LIN {X 0,Y 150.229,Z 301.582,A -85,B 0,C 180,E1 -24092.731,E2 -24092.731} C_VEL
LIN {X 0,Y 150.411,Z 301.529,A -85,B 0,C 180,E1 -24099.15,E2 -24099.15} C_VEL
LIN {X 0,Y 151.251,Z 301.453,A -85,B 0,C 180,E1 -24104.699,E2 -24104.699} C_VEL
LIN {X 0,Y 152.579,Z 314.488,A -85,B 0,C 180,E1 -24105.834,E2 -24105.834} C_VEL
LIN {X 0,Y 152.143,Z 366.9,A -85,B 0,C 180,E1 -24110.789,E2 -24110.789} C_VEL
LIN {X 0,Y 151.908,Z 379.421,A -85,B 0,C 180,E1 -24112.365,E2 -24112.365} C_VEL
LIN {X 0,Y 151.505,Z 390.839,A -85,B 0,C 180,E1 -24114.352,E2 -24114.352} C_VEL
LIN {X 0,Y 151.14,Z 401.236,A -85,B 0,C 180,E1 -24116.677,E2 -24116.677} C_VEL
LIN {X 0,Y 150.848,Z 410.602,A -85,B 0,C 180,E1 -24119.341,E2 -24119.341} C_VEL
LIN {X 0,Y 150.628,Z 416.487,A -85,B 0,C 180,E1 -24121.345,E2 -24121.345} C_VEL
LIN {X 0,Y 150.402,Z 424.552,A -85,B 0,C 180,E1 -24124.699,E2 -24124.699} C_VEL
LIN {X 0,Y 150.691,Z 431.338,A -85,B 0,C 180,E1 -24128.051,E2 -24128.051} C_VEL
LIN {X 0,Y 151.578,Z 437.961,A -85,B 0,C 180,E1 -24132.051,E2 -24132.051} C_VEL
LIN {X 0,Y 153.375,Z 443.251,A -85,B 0,C 180,E1 -24135.966,E2 -24135.966} C_VEL
LIN {X 0,Y 156.284,Z 447.464,A -85,B 0,C 180,E1 -24139.719,E2 -24139.719} C_VEL
LIN {X 0,Y 160.116,Z 450.667,A -85,B 0,C 180,E1 -24143.276,E2 -24143.276} C_VEL
LIN {X 0,Y 163.094,Z 452.341,A -85,B 0,C 180,E1 -24145.534,E2 -24145.534} C_VEL
LIN {X 0,Y 168.824,Z 454.022,A -85,B 0,C 180,E1 -24149.047,E2 -24149.047} C_VEL
LIN {X 0,Y 174.154,Z 454.577,A -85,B 0,C 180,E1 -24151.65,E2 -24151.65} C_VEL
LIN {X 0,Y 178.432,Z 454.52,A -85,B 0,C 180,E1 -24153.472,E2 -24153.472} C_VEL
LIN {X 0,Y 182.969,Z 453.929,A -85,B 0,C 180,E1 -24155.188,E2 -24155.188} C_VEL
LIN {X 0,Y 192.773,Z 451.539,A -85,B 0,C 180,E1 -24158.307,E2 -24158.307} C_VEL
LIN {X 0,Y 200.616,Z 448.43,A -85,B 0,C 180,E1 -24160.405,E2 -24160.405} C_VEL
LIN {X 0,Y 208.853,Z 444.151,A -85,B 0,C 180,E1 -24162.306,E2 -24162.306} C_VEL
LIN {X 0,Y 216.089,Z 439.514,A -85,B 0,C 180,E1 -24163.759,E2 -24163.759} C_VEL
LIN {X 0,Y 217.224,Z 438.727,A -85,B 0,C 180,E1 -24163.963,E2 -24163.963} C_VEL
LIN {X 0,Y 216.329,Z 439.432,A -85,B 0,C 180,E1 -24164.379,E2 -24164.379} C_VEL
LIN {X 0,Y 210.261,Z 443.858,A -85,B 0,C 180,E1 -24165.417,E2 -24165.417} C_VEL
LIN {X 0,Y 202.4,Z 448.708,A -85,B 0,C 180,E1 -24166.984,E2 -24166.984} C_VEL
LIN {X 0,Y 193.364,Z 453.242,A -85,B 0,C 180,E1 -24169.138,E2 -24169.138} C_VEL
LIN {X 0,Y 185.87,Z 456.12,A -85,B 0,C 180,E1 -24171.275,E2 -24171.275} C_VEL
LIN {X 0,Y 178.466,Z 458.224,A -85,B 0,C 180,E1 -24173.793,E2 -24173.793} C_VEL
LIN {X 0,Y 172.785,Z 459.125,A -85,B 0,C 180,E1 -24176.161,E2 -24176.161} C_VEL
LIN {X 0,Y 168.905,Z 459.398,A -85,B 0,C 180,E1 -24177.655,E2 -24177.655} C_VEL
LIN {X 0,Y 164.5,Z 459.233,A -85,B 0,C 180,E1 -24179.027,E2 -24179.027} C_VEL
LIN {X 0,Y 157.202,Z 458.002,A -85,B 0,C 180,E1 -24181.38,E2 -24181.38} C_VEL
LIN {X 0,Y 152.596,Z 456.474,A -85,B 0,C 180,E1 -24183.671,E2 -24183.671} C_VEL
LIN {X 0,Y 151.792,Z 455.973,A -85,B 0,C 180,E1 -24184.331,E2 -24184.331} C_VEL
LIN {X 0,Y 148.796,Z 453.802,A -85,B 0,C 180,E1 -24187.798,E2 -24187.798} C_VEL
LIN {X 0,Y 145.917,Z 449.099,A -85,B 0,C 180,E1 -24193.202,E2 -24193.202} C_VEL
LIN {X 0,Y 145.117,Z 445.833,A -85,B 0,C 180,E1 -24196.344,E2 -24196.344} C_VEL
LIN {X 0,Y 143.265,Z 449.83,A -85,B 0,C 180,E1 -24198.683,E2 -24198.683} C_VEL
LIN {X 0,Y 141.516,Z 455.368,A -85,B 0,C 180,E1 -24202.867,E2 -24202.867} C_VEL
LIN {X 0,Y 141.005,Z 459.469,A -85,B 0,C 180,E1 -24207.142,E2 -24207.142} C_VEL
LIN {X 0,Y 141.109,Z 461.507,A -85,B 0,C 180,E1 -24209.999,E2 -24209.999} C_VEL
LIN {X 0,Y 140.819,Z 463.144,A -85,B 0,C 180,E1 -24213.359,E2 -24213.359} C_VEL
LIN {X 0,Y 140.801,Z 463.878,A -85,B 0,C 180,E1 -24215.729,E2 -24215.729} C_VEL
LIN {X 0,Y 141.059,Z 464.25,A -85,B 0,C 180,E1 -24218.596,E2 -24218.596} C_VEL
LIN {X 0,Y 141.652,Z 464.181,A -85,B 0,C 180,E1 -24221.446,E2 -24221.446} C_VEL
LIN {X 0,Y 142.592,Z 463.67,A -85,B 0,C 180,E1 -24224.266,E2 -24224.266} C_VEL
LIN {X 0,Y 143.865,Z 462.646,A -85,B 0,C 180,E1 -24227.044,E2 -24227.044} C_VEL
LIN {X 0,Y 146.436,Z 460.124,A -85,B 0,C 180,E1 -24231.097,E2 -24231.097} C_VEL
LIN {X 0,Y 149.84,Z 456.335,A -85,B 0,C 180,E1 -24234.969,E2 -24234.969} C_VEL
LIN {X 0,Y 153.97,Z 451.2,A -85,B 0,C 180,E1 -24238.637,E2 -24238.637} C_VEL
LIN {X 0,Y 157.929,Z 445.711,A -85,B 0,C 180,E1 -24241.526,E2 -24241.526} C_VEL
LIN {X 0,Y 162.256,Z 438.889,A -85,B 0,C 180,E1 -24244.269,E2 -24244.269} C_VEL
LIN {X 0,Y 166.858,Z 430.459,A -85,B 0,C 180,E1 -24246.751,E2 -24246.751} C_VEL
LIN {X 0,Y 170.617,Z 422.486,A -85,B 0,C 180,E1 -24248.537,E2 -24248.537} C_VEL
LIN {X 0,Y 173.829,Z 414.514,A -85,B 0,C 180,E1 -24249.928,E2 -24249.928} C_VEL
LIN {X 0,Y 176.671,Z 406.274,A -85,B 0,C 180,E1 -24251.023,E2 -24251.023} C_VEL
LIN {X 0,Y 179.008,Z 397.922,A -85,B 0,C 180,E1 -24251.869,E2 -24251.869} C_VEL
LIN {X 0,Y 180.963,Z 388.209,A -85,B 0,C 180,E1 -24252.618,E2 -24252.618} C_VEL
LIN {X 0,Y 182.34,Z 377.856,A -85,B 0,C 180,E1 -24253.135,E2 -24253.135} C_VEL
LIN {X 0,Y 182.818,Z 371.037,A -85,B 0,C 180,E1 -24253.41,E2 -24253.41} C_VEL
LIN {X 0,Y 182.252,Z 365.36,A -85,B 0,C 180,E1 -24253.978,E2 -24253.978} C_VEL
LIN {X 0,Y 177.633,Z 353.901,A -85,B 0,C 180,E1 -24256.616,E2 -24256.616} C_VEL
LIN {X 0,Y 173.526,Z 345.27,A -85,B 0,C 180,E1 -24259.122,E2 -24259.122} C_VEL
LIN {X 0,Y 170.096,Z 338.97,A -85,B 0,C 180,E1 -24261.374,E2 -24261.374} C_VEL
LIN {X 0,Y 167.541,Z 334.457,A -85,B 0,C 180,E1 -24263.23,E2 -24263.23} C_VEL
LIN {X 0,Y 165.381,Z 330.639,A -85,B 0,C 180,E1 -24264.943,E2 -24264.943} C_VEL
LIN {X 0,Y 162.264,Z 325.564,A -85,B 0,C 180,E1 -24267.65,E2 -24267.65} C_VEL
LIN {X 0,Y 158.625,Z 320.076,A -85,B 0,C 180,E1 -24271.317,E2 -24271.317} C_VEL
LIN {X 0,Y 155.794,Z 317.621,A -85,B 0,C 180,E1 -24274.531,E2 -24274.531} C_VEL
LIN {X 0,Y 154.29,Z 314.613,A -85,B 0,C 180,E1 -24276.858,E2 -24276.858} C_VEL
LIN {X 0,Y 150.682,Z 311.854,A -85,B 0,C 180,E1 -24284.088,E2 -24284.088} C_VEL
LIN {X 0,Y 149.696,Z 308.547,A -85,B 0,C 180,E1 -24290.37,E2 -24290.37} C_VEL
LIN {X 0,Y 149.797,Z 308.81,A -85,B 0,C 180,E1 -24294.607,E2 -24294.607} C_VEL
LIN {X 0,Y 150.803,Z 310.633,A -85,B 0,C 180,E1 -24299.491,E2 -24299.491} C_VEL
LIN {X 0,Y 152.574,Z 313.389,A -85,B 0,C 180,E1 -24303.953,E2 -24303.953} C_VEL
LIN {X 0,Y 154.674,Z 314.736,A -85,B 0,C 180,E1 -24307.333,E2 -24307.333} C_VEL
LIN {X 0,Y 156.305,Z 317.841,A -85,B 0,C 180,E1 -24309.747,E2 -24309.747} C_VEL
LIN {X 0,Y 158.766,Z 320.202,A -85,B 0,C 180,E1 -24312.506,E2 -24312.506} C_VEL
LIN {X 0,Y 161.046,Z 323.638,A -85,B 0,C 180,E1 -24314.864,E2 -24314.864} C_VEL
LIN {X 0,Y 162.738,Z 325.43,A -85,B 0,C 180,E1 -24316.364,E2 -24316.364} C_VEL
LIN {X 0,Y 165.495,Z 329.24,A -85,B 0,C 180,E1 -24318.67,E2 -24318.67} C_VEL
LIN {X 0,Y 169.55,Z 335.043,A -85,B 0,C 180,E1 -24321.669,E2 -24321.669} C_VEL
LIN {X 0,Y 174.099,Z 341.826,A -85,B 0,C 180,E1 -24324.579,E2 -24324.579} C_VEL
LIN {X 0,Y 179.901,Z 351.582,A -85,B 0,C 180,E1 -24327.867,E2 -24327.867} C_VEL
LIN {X 0,Y 183.667,Z 358.715,A -85,B 0,C 180,E1 -24329.822,E2 -24329.822} C_VEL
LIN {X 0,Y 182.291,Z 374.31,A -85,B 0,C 180,E1 -24330.493,E2 -24330.493} C_VEL
LIN {X 0,Y 180.442,Z 384.951,A -85,B 0,C 180,E1 -24331.303,E2 -24331.303} C_VEL
LIN {X 0,Y 178.509,Z 393.196,A -85,B 0,C 180,E1 -24332.171,E2 -24332.171} C_VEL
LIN {X 0,Y 175.887,Z 401.994,A -85,B 0,C 180,E1 -24333.392,E2 -24333.392} C_VEL
LIN {X 0,Y 172.716,Z 410.391,A -85,B 0,C 180,E1 -24334.863,E2 -24334.863} C_VEL
LIN {X 0,Y 169.499,Z 417.801,A -85,B 0,C 180,E1 -24336.549,E2 -24336.549} C_VEL
LIN {X 0,Y 166.077,Z 424.565,A -85,B 0,C 180,E1 -24338.476,E2 -24338.476} C_VEL
LIN {X 0,Y 161.746,Z 431.819,A -85,B 0,C 180,E1 -24341.083,E2 -24341.083} C_VEL
LIN {X 0,Y 157.132,Z 438.434,A -85,B 0,C 180,E1 -24344.306,E2 -24344.306} C_VEL
LIN {X 0,Y 154.039,Z 442.386,A -85,B 0,C 180,E1 -24346.872,E2 -24346.872} C_VEL
LIN {X 0,Y 151.295,Z 445.463,A -85,B 0,C 180,E1 -24349.434,E2 -24349.434} C_VEL
LIN {X 0,Y 148.822,Z 447.877,A -85,B 0,C 180,E1 -24352.128,E2 -24352.128} C_VEL
LIN {X 0,Y 146.718,Z 449.672,A -85,B 0,C 180,E1 -24354.914,E2 -24354.914} C_VEL
LIN {X 0,Y 144.872,Z 450.906,A -85,B 0,C 180,E1 -24357.75,E2 -24357.75} C_VEL
LIN {X 0,Y 142.605,Z 451.785,A -85,B 0,C 180,E1 -24362.486,E2 -24362.486} C_VEL
LIN {X 0,Y 141.321,Z 451.399,A -85,B 0,C 180,E1 -24366.557,E2 -24366.557} C_VEL
LIN {X 0,Y 140.573,Z 449.331,A -85,B 0,C 180,E1 -24371.754,E2 -24371.754} C_VEL
LIN {X 0,Y 140.589,Z 446.8,A -85,B 0,C 180,E1 -24375.526,E2 -24375.526} C_VEL
LIN {X 0,Y 141.098,Z 442.555,A -85,B 0,C 180,E1 -24379.961,E2 -24379.961} C_VEL
LIN {X 0,Y 142.197,Z 436.794,A -85,B 0,C 180,E1 -24384.328,E2 -24384.328} C_VEL
LIN {X 0,Y 143.366,Z 430.499,A -85,B 0,C 180,E1 -24387.894,E2 -24387.894} C_VEL
LIN {X 0,Y 144.639,Z 424.336,A -85,B 0,C 180,E1 -24390.697,E2 -24390.697} C_VEL
LIN {X 0,Y 146.197,Z 416.829,A -85,B 0,C 180,E1 -24393.446,E2 -24393.446} C_VEL
LIN {X 0,Y 147.588,Z 410.023,A -85,B 0,C 180,E1 -24395.466,E2 -24395.466} C_VEL
LIN {X 0,Y 149.047,Z 401.938,A -85,B 0,C 180,E1 -24397.415,E2 -24397.415} C_VEL
LIN {X 0,Y 150.452,Z 393.174,A -85,B 0,C 180,E1 -24399.071,E2 -24399.071} C_VEL
LIN {X 0,Y 151.565,Z 383.214,A -85,B 0,C 180,E1 -24400.521,E2 -24400.521} C_VEL
LIN {X 0,Y 152.71,Z 370.439,A -85,B 0,C 180,E1 -24401.707,E2 -24401.707} C_VEL
LIN {X 0,Y 153.76,Z 346.37,A -85,B 0,C 180,E1 -24402.886,E2 -24402.886} C_VEL
LIN {X 0,Y 154.41,Z 327.759,A -85,B 0,C 180,E1 -24403.733,E2 -24403.733} C_VEL
LIN {X 0,Y 150.233,Z 317.497,A -85,B 0,C 180,E1 -24404.997,E2 -24404.997} C_VEL
LIN {X 0,Y 144.242,Z 305.25,A -85,B 0,C 180,E1 -24406.817,E2 -24406.817} C_VEL
LIN {X 0,Y 143.241,Z 302.455,A -85,B 0,C 180,E1 -24407.213,E2 -24407.213} C_VEL
LIN {X 0,Y 143.249,Z 302.455,A -85,B 0,C 180,E1 -24411.256,E2 -24411.256} C_VEL
LIN {X 0,Y 143.159,Z 302.465,A -85,B 0,C 180,E1 -24417.936,E2 -24417.936} C_VEL
LIN {X 0,Y 143.113,Z 302.461,A -85,B 0,C 180,E1 -24423.421,E2 -24423.421} C_VEL
LIN {X 0,Y 143.032,Z 302.477,A -85,B 0,C 180,E1 -24429.701,E2 -24429.701} C_VEL
LIN {X 0,Y 143.014,Z 302.478,A -85,B 0,C 180,E1 -24433.472,E2 -24433.472} C_VEL
LIN {X 0,Y 143.022,Z 302.482,A -85,B 0,C 180,E1 -24437.485,E2 -24437.485} C_VEL
LIN {X 0,Y 143.06,Z 302.473,A -85,B 0,C 180,E1 -24441.816,E2 -24441.816} C_VEL
LIN {X 0,Y 143.164,Z 302.459,A -85,B 0,C 180,E1 -24447.329,E2 -24447.329} C_VEL
LIN {X 0,Y 143.146,Z 302.462,A -85,B 0,C 180,E1 -24453.788,E2 -24453.788} C_VEL
LIN {X 0,Y 143.414,Z 302.402,A -85,B 0,C 180,E1 -24459.948,E2 -24459.948} C_VEL
LIN {X 0,Y 144.372,Z 302.313,A -85,B 0,C 180,E1 -24465.33,E2 -24465.33} C_VEL
LIN {X 0,Y 145.649,Z 314.508,A -85,B 0,C 180,E1 -24466.404,E2 -24466.404} C_VEL
LIN {X 0,Y 145.428,Z 365.822,A -85,B 0,C 180,E1 -24471.586,E2 -24471.586} C_VEL
LIN {X 0,Y 145.209,Z 378.736,A -85,B 0,C 180,E1 -24473.234,E2 -24473.234} C_VEL
LIN {X 0,Y 144.862,Z 389.408,A -85,B 0,C 180,E1 -24475.139,E2 -24475.139} C_VEL
LIN {X 0,Y 144.515,Z 400.112,A -85,B 0,C 180,E1 -24477.57,E2 -24477.57} C_VEL
LIN {X 0,Y 144.262,Z 410.585,A -85,B 0,C 180,E1 -24480.707,E2 -24480.707} C_VEL
LIN {X 0,Y 143.969,Z 418.075,A -85,B 0,C 180,E1 -24483.507,E2 -24483.507} C_VEL
LIN {X 0,Y 143.94,Z 425.928,A -85,B 0,C 180,E1 -24487.02,E2 -24487.02} C_VEL
LIN {X 0,Y 144.613,Z 433.562,A -85,B 0,C 180,E1 -24491.218,E2 -24491.218} C_VEL
LIN {X 0,Y 146.4,Z 440.494,A -85,B 0,C 180,E1 -24495.958,E2 -24495.958} C_VEL
LIN {X 0,Y 148.706,Z 444.681,A -85,B 0,C 180,E1 -24499.327,E2 -24499.327} C_VEL
LIN {X 0,Y 152.233,Z 448.67,A -85,B 0,C 180,E1 -24503.113,E2 -24503.113} C_VEL
LIN {X 0,Y 156.758,Z 451.664,A -85,B 0,C 180,E1 -24506.645,E2 -24506.645} C_VEL
LIN {X 0,Y 163.972,Z 454.29,A -85,B 0,C 180,E1 -24510.961,E2 -24510.961} C_VEL
LIN {X 0,Y 172.553,Z 455.098,A -85,B 0,C 180,E1 -24514.773,E2 -24514.773} C_VEL
LIN {X 0,Y 177.248,Z 454.952,A -85,B 0,C 180,E1 -24516.503,E2 -24516.503} C_VEL
LIN {X 0,Y 182.189,Z 454.309,A -85,B 0,C 180,E1 -24518.12,E2 -24518.12} C_VEL
LIN {X 0,Y 187.345,Z 453.182,A -85,B 0,C 180,E1 -24519.63,E2 -24519.63} C_VEL
LIN {X 0,Y 198.186,Z 449.699,A -85,B 0,C 180,E1 -24522.366,E2 -24522.366} C_VEL
LIN {X 0,Y 203.871,Z 447.147,A -85,B 0,C 180,E1 -24523.594,E2 -24523.594} C_VEL
LIN {X 0,Y 205.328,Z 446.454,A -85,B 0,C 180,E1 -24524.044,E2 -24524.044} C_VEL
LIN {X 0,Y 195.558,Z 451.445,A -85,B 0,C 180,E1 -24525.96,E2 -24525.96} C_VEL
LIN {X 0,Y 188.075,Z 454.463,A -85,B 0,C 180,E1 -24527.729,E2 -24527.729} C_VEL
LIN {X 0,Y 182.737,Z 456.222,A -85,B 0,C 180,E1 -24529.17,E2 -24529.17} C_VEL
LIN {X 0,Y 172.779,Z 458.32,A -85,B 0,C 180,E1 -24532.399,E2 -24532.399} C_VEL
LIN {X 0,Y 167.077,Z 458.858,A -85,B 0,C 180,E1 -24534.749,E2 -24534.749} C_VEL
LIN {X 0,Y 160.228,Z 458.587,A -85,B 0,C 180,E1 -24538.24,E2 -24538.24} C_VEL
LIN {X 0,Y 156.703,Z 457.974,A -85,B 0,C 180,E1 -24540.439,E2 -24540.439} C_VEL
LIN {X 0,Y 151.792,Z 455.973,A -85,B 0,C 180,E1 -24544.331,E2 -24544.331} C_VEL
LIN {X 0,Y 149.289,Z 454.599,A -85,B 0,C 180,E1 -24546.289,E2 -24546.289} C_VEL
LIN {X 0,Y 144.403,Z 451.099,A -85,B 0,C 180,E1 -24549.353,E2 -24549.353} C_VEL
LIN {X 0,Y 140.942,Z 447.628,A -85,B 0,C 180,E1 -24551.881,E2 -24551.881} C_VEL
LIN {X 0,Y 139.307,Z 444.952,A -85,B 0,C 180,E1 -24553.944,E2 -24553.944} C_VEL
LIN {X 0,Y 139.045,Z 444.062,A -85,B 0,C 180,E1 -24554.673,E2 -24554.673} C_VEL
LIN {X 0,Y 138.869,Z 443.792,A -85,B 0,C 180,E1 -24555.071,E2 -24555.071} C_VEL
LIN {X 0,Y 135.966,Z 450.073,A -85,B 0,C 180,E1 -24558.823,E2 -24558.823} C_VEL
LIN {X 0,Y 134.504,Z 454.69,A -85,B 0,C 180,E1 -24562.493,E2 -24562.493} C_VEL
LIN {X 0,Y 133.922,Z 458.874,A -85,B 0,C 180,E1 -24566.991,E2 -24566.991} C_VEL
LIN {X 0,Y 134.022,Z 460.991,A -85,B 0,C 180,E1 -24569.999,E2 -24569.999} C_VEL
LIN {X 0,Y 133.753,Z 462.578,A -85,B 0,C 180,E1 -24573.164,E2 -24573.164} C_VEL
LIN {X 0,Y 133.731,Z 463.437,A -85,B 0,C 180,E1 -24576.033,E2 -24576.033} C_VEL
LIN {X 0,Y 134.047,Z 463.884,A -85,B 0,C 180,E1 -24579.049,E2 -24579.049} C_VEL
LIN {X 0,Y 134.703,Z 463.891,A -85,B 0,C 180,E1 -24582.045,E2 -24582.045} C_VEL
LIN {X 0,Y 135.695,Z 463.451,A -85,B 0,C 180,E1 -24585.008,E2 -24585.008} C_VEL
LIN {X 0,Y 137.063,Z 462.441,A -85,B 0,C 180,E1 -24587.917,E2 -24587.917} C_VEL
LIN {X 0,Y 139.822,Z 460.061,A -85,B 0,C 180,E1 -24592.146,E2 -24592.146} C_VEL
LIN {X 0,Y 143.446,Z 456.388,A -85,B 0,C 180,E1 -24596.164,E2 -24596.164} C_VEL
LIN {X 0,Y 146.252,Z 453.266,A -85,B 0,C 180,E1 -24598.72,E2 -24598.72} C_VEL
LIN {X 0,Y 150.204,Z 448.323,A -85,B 0,C 180,E1 -24601.761,E2 -24601.761} C_VEL
LIN {X 0,Y 154.607,Z 442.118,A -85,B 0,C 180,E1 -24604.625,E2 -24604.625} C_VEL
LIN {X 0,Y 158.342,Z 436.234,A -85,B 0,C 180,E1 -24606.74,E2 -24606.74} C_VEL
LIN {X 0,Y 162.494,Z 428.754,A -85,B 0,C 180,E1 -24608.84,E2 -24608.84} C_VEL
LIN {X 0,Y 166.254,Z 420.938,A -85,B 0,C 180,E1 -24610.537,E2 -24610.537} C_VEL
LIN {X 0,Y 169.609,Z 412.703,A -85,B 0,C 180,E1 -24611.925,E2 -24611.925} C_VEL
LIN {X 0,Y 173.221,Z 402.214,A -85,B 0,C 180,E1 -24613.208,E2 -24613.208} C_VEL
LIN {X 0,Y 175.97,Z 390.544,A -85,B 0,C 180,E1 -24614.209,E2 -24614.209} C_VEL
LIN {X 0,Y 177.455,Z 381.277,A -85,B 0,C 180,E1 -24614.735,E2 -24614.735} C_VEL
LIN {X 0,Y 178.245,Z 371.665,A -85,B 0,C 180,E1 -24615.169,E2 -24615.169} C_VEL
LIN {X 0,Y 177.929,Z 368.636,A -85,B 0,C 180,E1 -24615.5,E2 -24615.5} C_VEL
LIN {X 0,Y 173.611,Z 357.538,A -85,B 0,C 180,E1 -24618.181,E2 -24618.181} C_VEL
LIN {X 0,Y 168.856,Z 347.52,A -85,B 0,C 180,E1 -24621.36,E2 -24621.36} C_VEL
LIN {X 0,Y 165.244,Z 340.753,A -85,B 0,C 180,E1 -24624.095,E2 -24624.095} C_VEL
LIN {X 0,Y 162.708,Z 336.151,A -85,B 0,C 180,E1 -24626.239,E2 -24626.239} C_VEL
LIN {X 0,Y 159.969,Z 331.576,A -85,B 0,C 180,E1 -24628.797,E2 -24628.797} C_VEL
LIN {X 0,Y 156.838,Z 326.655,A -85,B 0,C 180,E1 -24632.173,E2 -24632.173} C_VEL
LIN {X 0,Y 154.322,Z 324.345,A -85,B 0,C 180,E1 -24635.202,E2 -24635.202} C_VEL
LIN {X 0,Y 152.819,Z 321.374,A -85,B 0,C 180,E1 -24637.695,E2 -24637.695} C_VEL
LIN {X 0,Y 149.61,Z 318.707,A -85,B 0,C 180,E1 -24644.67,E2 -24644.67} C_VEL
LIN {X 0,Y 148.808,Z 315.59,A -85,B 0,C 180,E1 -24650.476,E2 -24650.476} C_VEL
LIN {X 0,Y 148.867,Z 315.755,A -85,B 0,C 180,E1 -24654.122,E2 -24654.122} C_VEL
LIN {X 0,Y 149.747,Z 317.562,A -85,B 0,C 180,E1 -24658.983,E2 -24658.983} C_VEL
LIN {X 0,Y 151.67,Z 320.5,A -85,B 0,C 180,E1 -24663.977,E2 -24663.977} C_VEL
LIN {X 0,Y 153.228,Z 321.507,A -85,B 0,C 180,E1 -24666.576,E2 -24666.576} C_VEL
LIN {X 0,Y 155.002,Z 324.786,A -85,B 0,C 180,E1 -24669.33,E2 -24669.33} C_VEL
LIN {X 0,Y 157.037,Z 326.851,A -85,B 0,C 180,E1 -24671.724,E2 -24671.724} C_VEL
LIN {X 0,Y 159.682,Z 330.667,A -85,B 0,C 180,E1 -24674.541,E2 -24674.541} C_VEL
LIN {X 0,Y 160.757,Z 331.914,A -85,B 0,C 180,E1 -24675.541,E2 -24675.541} C_VEL
LIN {X 0,Y 164.328,Z 337.057,A -85,B 0,C 180,E1 -24678.632,E2 -24678.632} C_VEL
LIN {X 0,Y 168.845,Z 343.724,A -85,B 0,C 180,E1 -24681.991,E2 -24681.991} C_VEL
LIN {X 0,Y 174.488,Z 353.184,A -85,B 0,C 180,E1 -24685.592,E2 -24685.592} C_VEL
LIN {X 0,Y 179.07,Z 361.751,A -85,B 0,C 180,E1 -24688.193,E2 -24688.193} C_VEL
LIN {X 0,Y 177.537,Z 376.056,A -85,B 0,C 180,E1 -24688.844,E2 -24688.844} C_VEL
LIN {X 0,Y 175.55,Z 386.635,A -85,B 0,C 180,E1 -24689.696,E2 -24689.696} C_VEL
LIN {X 0,Y 173.269,Z 395.493,A -85,B 0,C 180,E1 -24690.685,E2 -24690.685} C_VEL
LIN {X 0,Y 170.098,Z 405.083,A -85,B 0,C 180,E1 -24692.1,E2 -24692.1} C_VEL
LIN {X 0,Y 165.668,Z 415.577,A -85,B 0,C 180,E1 -24694.185,E2 -24694.185} C_VEL
LIN {X 0,Y 161.476,Z 423.654,A -85,B 0,C 180,E1 -24696.373,E2 -24696.373} C_VEL
LIN {X 0,Y 157.661,Z 430.042,A -85,B 0,C 180,E1 -24698.602,E2 -24698.602} C_VEL
LIN {X 0,Y 153.779,Z 435.622,A -85,B 0,C 180,E1 -24701.055,E2 -24701.055} C_VEL
LIN {X 0,Y 150.313,Z 440.064,A -85,B 0,C 180,E1 -24703.555,E2 -24703.555} C_VEL
LIN {X 0,Y 146.858,Z 444.005,A -85,B 0,C 180,E1 -24706.434,E2 -24706.434} C_VEL
LIN {X 0,Y 142.981,Z 447.799,A -85,B 0,C 180,E1 -24710.284,E2 -24710.284} C_VEL
LIN {X 0,Y 140.641,Z 449.719,A -85,B 0,C 180,E1 -24713.155,E2 -24713.155} C_VEL
LIN {X 0,Y 138.588,Z 451.073,A -85,B 0,C 180,E1 -24716.095,E2 -24716.095} C_VEL
LIN {X 0,Y 136.905,Z 451.89,A -85,B 0,C 180,E1 -24719.113,E2 -24719.113} C_VEL
LIN {X 0,Y 135.549,Z 452.155,A -85,B 0,C 180,E1 -24722.184,E2 -24722.184} C_VEL
LIN {X 0,Y 134.516,Z 451.806,A -85,B 0,C 180,E1 -24725.294,E2 -24725.294} C_VEL
LIN {X 0,Y 133.837,Z 450.922,A -85,B 0,C 180,E1 -24728.434,E2 -24728.434} C_VEL
LIN {X 0,Y 133.489,Z 449.515,A -85,B 0,C 180,E1 -24731.586,E2 -24731.586} C_VEL
LIN {X 0,Y 133.546,Z 446.35,A -85,B 0,C 180,E1 -24736.302,E2 -24736.302} C_VEL
LIN {X 0,Y 134.164,Z 441.844,A -85,B 0,C 180,E1 -24740.959,E2 -24740.959} C_VEL
LIN {X 0,Y 135.196,Z 436.786,A -85,B 0,C 180,E1 -24744.781,E2 -24744.781} C_VEL
LIN {X 0,Y 136.436,Z 430.418,A -85,B 0,C 180,E1 -24748.525,E2 -24748.525} C_VEL
LIN {X 0,Y 137.805,Z 424.172,A -85,B 0,C 180,E1 -24751.462,E2 -24751.462} C_VEL
LIN {X 0,Y 139.219,Z 417.615,A -85,B 0,C 180,E1 -24753.981,E2 -24753.981} C_VEL
LIN {X 0,Y 140.855,Z 409.977,A -85,B 0,C 180,E1 -24756.352,E2 -24756.352} C_VEL
LIN {X 0,Y 142.479,Z 401.257,A -85,B 0,C 180,E1 -24758.51,E2 -24758.51} C_VEL
LIN {X 0,Y 143.928,Z 392.452,A -85,B 0,C 180,E1 -24760.196,E2 -24760.196} C_VEL
LIN {X 0,Y 145.344,Z 380.299,A -85,B 0,C 180,E1 -24761.894,E2 -24761.894} C_VEL
LIN {X 0,Y 146.214,Z 369.812,A -85,B 0,C 180,E1 -24762.809,E2 -24762.809} C_VEL
LIN {X 0,Y 147.991,Z 329.484,A -85,B 0,C 180,E1 -24764.764,E2 -24764.764} C_VEL
LIN {X 0,Y 143.545,Z 318.841,A -85,B 0,C 180,E1 -24766.196,E2 -24766.196} C_VEL
LIN {X 0,Y 137.281,Z 306.261,A -85,B 0,C 180,E1 -24768.256,E2 -24768.256} C_VEL
LIN {X 0,Y 136.24,Z 303.326,A -85,B 0,C 180,E1 -24768.713,E2 -24768.713} C_VEL
LIN {X 0,Y 136.17,Z 303.337,A -85,B 0,C 180,E1 -24771.749,E2 -24771.749} C_VEL
LIN {X 0,Y 136.068,Z 303.348,A -85,B 0,C 180,E1 -24778.615,E2 -24778.615} C_VEL
LIN {X 0,Y 136.018,Z 303.35,A -85,B 0,C 180,E1 -24784.637,E2 -24784.637} C_VEL
LIN {X 0,Y 136.004,Z 303.35,A -85,B 0,C 180,E1 -24789.201,E2 -24789.201} C_VEL
LIN {X 0,Y 135.959,Z 303.356,A -85,B 0,C 180,E1 -24793.656,E2 -24793.656} C_VEL
LIN {X 0,Y 135.967,Z 303.361,A -85,B 0,C 180,E1 -24797.797,E2 -24797.797} C_VEL
LIN {X 0,Y 136.009,Z 303.35,A -85,B 0,C 180,E1 -24801.692,E2 -24801.692} C_VEL
LIN {X 0,Y 136.04,Z 303.35,A -85,B 0,C 180,E1 -24805.75,E2 -24805.75} C_VEL
LIN {X 0,Y 136.13,Z 303.339,A -85,B 0,C 180,E1 -24812.325,E2 -24812.325} C_VEL
LIN {X 0,Y 136.292,Z 303.286,A -85,B 0,C 180,E1 -24818.852,E2 -24818.852} C_VEL
LIN {X 0,Y 137.563,Z 303.366,A -85,B 0,C 180,E1 -24826.097,E2 -24826.097} C_VEL
LIN {X 0,Y 138.771,Z 314.19,A -85,B 0,C 180,E1 -24827.085,E2 -24827.085} C_VEL
LIN {X 0,Y 138.755,Z 364.726,A -85,B 0,C 180,E1 -24832.461,E2 -24832.461} C_VEL
LIN {X 0,Y 138.569,Z 377.937,A -85,B 0,C 180,E1 -24834.188,E2 -24834.188} C_VEL
LIN {X 0,Y 138.272,Z 389.442,A -85,B 0,C 180,E1 -24836.367,E2 -24836.367} C_VEL
LIN {X 0,Y 138.024,Z 398.544,A -85,B 0,C 180,E1 -24838.551,E2 -24838.551} C_VEL
LIN {X 0,Y 137.761,Z 409.444,A -85,B 0,C 180,E1 -24841.837,E2 -24841.837} C_VEL
LIN {X 0,Y 137.442,Z 417.832,A -85,B 0,C 180,E1 -24845.143,E2 -24845.143} C_VEL
LIN {X 0,Y 137.658,Z 425.577,A -85,B 0,C 180,E1 -24848.819,E2 -24848.819} C_VEL
LIN {X 0,Y 138.46,Z 433.274,A -85,B 0,C 180,E1 -24853.213,E2 -24853.213} C_VEL
LIN {X 0,Y 140.874,Z 440.628,A -85,B 0,C 180,E1 -24858.423,E2 -24858.423} C_VEL
LIN {X 0,Y 143.277,Z 444.571,A -85,B 0,C 180,E1 -24861.594,E2 -24861.594} C_VEL
LIN {X 0,Y 147.322,Z 448.626,A -85,B 0,C 180,E1 -24865.435,E2 -24865.435} C_VEL
LIN {X 0,Y 150.494,Z 450.887,A -85,B 0,C 180,E1 -24867.848,E2 -24867.848} C_VEL
LIN {X 0,Y 154.042,Z 452.618,A -85,B 0,C 180,E1 -24870.132,E2 -24870.132} C_VEL
LIN {X 0,Y 158.157,Z 454.02,A -85,B 0,C 180,E1 -24872.402,E2 -24872.402} C_VEL
LIN {X 0,Y 162.227,Z 454.98,A -85,B 0,C 180,E1 -24874.285,E2 -24874.285} C_VEL
LIN {X 0,Y 166.771,Z 455.541,A -85,B 0,C 180,E1 -24876.164,E2 -24876.164} C_VEL
LIN {X 0,Y 176.67,Z 455.363,A -85,B 0,C 180,E1 -24879.538,E2 -24879.538} C_VEL
LIN {X 0,Y 181.997,Z 454.684,A -85,B 0,C 180,E1 -24881.039,E2 -24881.039} C_VEL
LIN {X 0,Y 187.484,Z 453.476,A -85,B 0,C 180,E1 -24882.442,E2 -24882.442} C_VEL
LIN {X 0,Y 193.113,Z 451.843,A -85,B 0,C 180,E1 -24883.754,E2 -24883.754} C_VEL
LIN {X 0,Y 190.934,Z 452.748,A -85,B 0,C 180,E1 -24884.383,E2 -24884.383} C_VEL
LIN {X 0,Y 182.872,Z 455.41,A -85,B 0,C 180,E1 -24886.23,E2 -24886.23} C_VEL
LIN {X 0,Y 172.168,Z 457.669,A -85,B 0,C 180,E1 -24889.221,E2 -24889.221} C_VEL
LIN {X 0,Y 167.203,Z 458.232,A -85,B 0,C 180,E1 -24890.913,E2 -24890.913} C_VEL
LIN {X 0,Y 158.263,Z 458.132,A -85,B 0,C 180,E1 -24894.739,E2 -24894.739} C_VEL
LIN {X 0,Y 154.298,Z 457.571,A -85,B 0,C 180,E1 -24896.867,E2 -24896.867} C_VEL
LIN {X 0,Y 147.42,Z 455.286,A -85,B 0,C 180,E1 -24901.527,E2 -24901.527} C_VEL
LIN {X 0,Y 143.568,Z 452.688,A -85,B 0,C 180,E1 -24905.411,E2 -24905.411} C_VEL
LIN {X 0,Y 140.851,Z 449.275,A -85,B 0,C 180,E1 -24909.556,E2 -24909.556} C_VEL
LIN {X 0,Y 139.328,Z 445.437,A -85,B 0,C 180,E1 -24913.441,E2 -24913.441} C_VEL
LIN {X 0,Y 139.045,Z 444.062,A -85,B 0,C 180,E1 -24914.673,E2 -24914.673} C_VEL
LIN {X 0,Y 138.762,Z 444.37,A -85,B 0,C 180,E1 -24915.346,E2 -24915.346} C_VEL
LIN {X 0,Y 137.507,Z 446.848,A -85,B 0,C 180,E1 -24916.8,E2 -24916.8} C_VEL
LIN {X 0,Y 134.856,Z 449.882,A -85,B 0,C 180,E1 -24918.686,E2 -24918.686} C_VEL
LIN {X 0,Y 128.597,Z 455.232,A -85,B 0,C 180,E1 -24922.917,E2 -24922.917} C_VEL
LIN {X 0,Y 127.121,Z 456.775,A -85,B 0,C 180,E1 -24924.91,E2 -24924.91} C_VEL
LIN {X 0,Y 126.913,Z 457.415,A -85,B 0,C 180,E1 -24925.745,E2 -24925.745} C_VEL
LIN {X 0,Y 126.937,Z 460.465,A -85,B 0,C 180,E1 -24929.999,E2 -24929.999} C_VEL
LIN {X 0,Y 126.677,Z 462.009,A -85,B 0,C 180,E1 -24933.18,E2 -24933.18} C_VEL
LIN {X 0,Y 126.69,Z 462.989,A -85,B 0,C 180,E1 -24936.369,E2 -24936.369} C_VEL
LIN {X 0,Y 127.033,Z 463.515,A -85,B 0,C 180,E1 -24939.553,E2 -24939.553} C_VEL
LIN {X 0,Y 127.744,Z 463.602,A -85,B 0,C 180,E1 -24942.712,E2 -24942.712} C_VEL
LIN {X 0,Y 128.823,Z 463.205,A -85,B 0,C 180,E1 -24945.829,E2 -24945.829} C_VEL
LIN {X 0,Y 130.297,Z 462.233,A -85,B 0,C 180,E1 -24948.882,E2 -24948.882} C_VEL
LIN {X 0,Y 132.143,Z 460.796,A -85,B 0,C 180,E1 -24951.857,E2 -24951.857} C_VEL
LIN {X 0,Y 135.728,Z 457.71,A -85,B 0,C 180,E1 -24956.112,E2 -24956.112} C_VEL
LIN {X 0,Y 140.06,Z 453.37,A -85,B 0,C 180,E1 -24960.117,E2 -24960.117} C_VEL
LIN {X 0,Y 145.127,Z 447.409,A -85,B 0,C 180,E1 -24963.842,E2 -24963.842} C_VEL
LIN {X 0,Y 148.842,Z 442.501,A -85,B 0,C 180,E1 -24966.172,E2 -24966.172} C_VEL
LIN {X 0,Y 153.285,Z 435.886,A -85,B 0,C 180,E1 -24968.595,E2 -24968.595} C_VEL
LIN {X 0,Y 157.587,Z 428.44,A -85,B 0,C 180,E1 -24970.709,E2 -24970.709} C_VEL
LIN {X 0,Y 161.533,Z 420.614,A -85,B 0,C 180,E1 -24972.405,E2 -24972.405} C_VEL
LIN {X 0,Y 165.033,Z 412.379,A -85,B 0,C 180,E1 -24973.789,E2 -24973.789} C_VEL
LIN {X 0,Y 168.779,Z 401.889,A -85,B 0,C 180,E1 -24975.062,E2 -24975.062} C_VEL
LIN {X 0,Y 171.557,Z 390.601,A -85,B 0,C 180,E1 -24976.034,E2 -24976.034} C_VEL
LIN {X 0,Y 173.14,Z 381.093,A -85,B 0,C 180,E1 -24976.58,E2 -24976.58} C_VEL
LIN {X 0,Y 173.872,Z 372.692,A -85,B 0,C 180,E1 -24976.98,E2 -24976.98} C_VEL
LIN {X 0,Y 172.172,Z 367.45,A -85,B 0,C 180,E1 -24978.141,E2 -24978.141} C_VEL
LIN {X 0,Y 168.483,Z 358.462,A -85,B 0,C 180,E1 -24980.681,E2 -24980.681} C_VEL
LIN {X 0,Y 164.76,Z 350.641,A -85,B 0,C 180,E1 -24983.503,E2 -24983.503} C_VEL
LIN {X 0,Y 161.618,Z 344.44,A -85,B 0,C 180,E1 -24986.185,E2 -24986.185} C_VEL
LIN {X 0,Y 158.239,Z 338.231,A -85,B 0,C 180,E1 -24989.472,E2 -24989.472} C_VEL
LIN {X 0,Y 155.089,Z 333.244,A -85,B 0,C 180,E1 -24993.045,E2 -24993.045} C_VEL
LIN {X 0,Y 152.685,Z 330.72,A -85,B 0,C 180,E1 -24996.19,E2 -24996.19} C_VEL
LIN {X 0,Y 151.364,Z 328.169,A -85,B 0,C 180,E1 -24998.562,E2 -24998.562} C_VEL
LIN {X 0,Y 148.467,Z 325.376,A -85,B 0,C 180,E1 -25005.602,E2 -25005.602} C_VEL
LIN {X 0,Y 147.909,Z 322.758,A -85,B 0,C 180,E1 -25010.417,E2 -25010.417} C_VEL
LIN {X 0,Y 147.973,Z 322.852,A -85,B 0,C 180,E1 -25014.13,E2 -25014.13} C_VEL
LIN {X 0,Y 148.699,Z 324.483,A -85,B 0,C 180,E1 -25018.468,E2 -25018.468} C_VEL
LIN {X 0,Y 150.596,Z 327.471,A -85,B 0,C 180,E1 -25023.67,E2 -25023.67} C_VEL
LIN {X 0,Y 151.898,Z 328.45,A -85,B 0,C 180,E1 -25025.967,E2 -25025.967} C_VEL
LIN {X 0,Y 153.833,Z 331.865,A -85,B 0,C 180,E1 -25029.07,E2 -25029.07} C_VEL
LIN {X 0,Y 155.386,Z 333.564,A -85,B 0,C 180,E1 -25030.983,E2 -25030.983} C_VEL
LIN {X 0,Y 158.09,Z 337.408,A -85,B 0,C 180,E1 -25033.98,E2 -25033.98} C_VEL
LIN {X 0,Y 162.046,Z 343.193,A -85,B 0,C 180,E1 -25037.664,E2 -25037.664} C_VEL
LIN {X 0,Y 166.202,Z 349.629,A -85,B 0,C 180,E1 -25040.956,E2 -25040.956} C_VEL
LIN {X 0,Y 171.155,Z 358.225,A -85,B 0,C 180,E1 -25044.357,E2 -25044.357} C_VEL
LIN {X 0,Y 174.553,Z 364.68,A -85,B 0,C 180,E1 -25046.44,E2 -25046.44} C_VEL
LIN {X 0,Y 173.131,Z 376.829,A -85,B 0,C 180,E1 -25047.053,E2 -25047.053} C_VEL
LIN {X 0,Y 171.138,Z 386.877,A -85,B 0,C 180,E1 -25047.855,E2 -25047.855} C_VEL
LIN {X 0,Y 168.961,Z 395.137,A -85,B 0,C 180,E1 -25048.771,E2 -25048.771} C_VEL
LIN {X 0,Y 166.248,Z 403.283,A -85,B 0,C 180,E1 -25049.932,E2 -25049.932} C_VEL
LIN {X 0,Y 162.716,Z 411.765,A -85,B 0,C 180,E1 -25051.457,E2 -25051.457} C_VEL
LIN {X 0,Y 158.812,Z 419.777,A -85,B 0,C 180,E1 -25053.355,E2 -25053.355} C_VEL
LIN {X 0,Y 154.276,Z 427.67,A -85,B 0,C 180,E1 -25055.786,E2 -25055.786} C_VEL
LIN {X 0,Y 148.976,Z 435.108,A -85,B 0,C 180,E1 -25058.887,E2 -25058.887} C_VEL
LIN {X 0,Y 145.26,Z 439.708,A -85,B 0,C 180,E1 -25061.417,E2 -25061.417} C_VEL
LIN {X 0,Y 142.205,Z 443.129,A -85,B 0,C 180,E1 -25063.766,E2 -25063.766} C_VEL
LIN {X 0,Y 138.733,Z 446.535,A -85,B 0,C 180,E1 -25066.852,E2 -25066.852} C_VEL
LIN {X 0,Y 134.704,Z 449.767,A -85,B 0,C 180,E1 -25071.239,E2 -25071.239} C_VEL
LIN {X 0,Y 132.449,Z 451.24,A -85,B 0,C 180,E1 -25074.291,E2 -25074.291} C_VEL
LIN {X 0,Y 130.523,Z 452.159,A -85,B 0,C 180,E1 -25077.423,E2 -25077.423} C_VEL
LIN {X 0,Y 128.993,Z 452.459,A -85,B 0,C 180,E1 -25080.637,E2 -25080.637} C_VEL
LIN {X 0,Y 127.772,Z 452.206,A -85,B 0,C 180,E1 -25083.895,E2 -25083.895} C_VEL
LIN {X 0,Y 126.949,Z 451.438,A -85,B 0,C 180,E1 -25087.2,E2 -25087.2} C_VEL
LIN {X 0,Y 126.448,Z 449.98,A -85,B 0,C 180,E1 -25090.847,E2 -25090.847} C_VEL
LIN {X 0,Y 126.387,Z 447.103,A -85,B 0,C 180,E1 -25095.509,E2 -25095.509} C_VEL
LIN {X 0,Y 126.688,Z 444.33,A -85,B 0,C 180,E1 -25098.805,E2 -25098.805} C_VEL
LIN {X 0,Y 127.71,Z 438.921,A -85,B 0,C 180,E1 -25103.682,E2 -25103.682} C_VEL
LIN {X 0,Y 129.24,Z 431.743,A -85,B 0,C 180,E1 -25108.443,E2 -25108.443} C_VEL
LIN {X 0,Y 130.582,Z 425.703,A -85,B 0,C 180,E1 -25111.543,E2 -25111.543} C_VEL
LIN {X 0,Y 132.262,Z 418.336,A -85,B 0,C 180,E1 -25114.572,E2 -25114.572} C_VEL
LIN {X 0,Y 133.808,Z 411.457,A -85,B 0,C 180,E1 -25116.863,E2 -25116.863} C_VEL
LIN {X 0,Y 135.413,Z 403.672,A -85,B 0,C 180,E1 -25118.958,E2 -25118.958} C_VEL
LIN {X 0,Y 136.914,Z 395.375,A -85,B 0,C 180,E1 -25120.725,E2 -25120.725} C_VEL
LIN {X 0,Y 138.113,Z 386.212,A -85,B 0,C 180,E1 -25122.248,E2 -25122.248} C_VEL
LIN {X 0,Y 139.321,Z 375.322,A -85,B 0,C 180,E1 -25123.517,E2 -25123.517} C_VEL
LIN {X 0,Y 140.184,Z 361.173,A -85,B 0,C 180,E1 -25124.453,E2 -25124.453} C_VEL
LIN {X 0,Y 141.5,Z 331.054,A -85,B 0,C 180,E1 -25125.913,E2 -25125.913} C_VEL
LIN {X 0,Y 136.093,Z 318.478,A -85,B 0,C 180,E1 -25127.786,E2 -25127.786} C_VEL
LIN {X 0,Y 130.179,Z 307.069,A -85,B 0,C 180,E1 -25129.905,E2 -25129.905} C_VEL
LIN {X 0,Y 129.166,Z 304.207,A -85,B 0,C 180,E1 -25130.444,E2 -25130.444} C_VEL
LIN {X 0,Y 128.999,Z 304.228,A -85,B 0,C 180,E1 -25135.84,E2 -25135.84} C_VEL
LIN {X 0,Y 128.994,Z 304.224,A -85,B 0,C 180,E1 -25139.364,E2 -25139.364} C_VEL
LIN {X 0,Y 128.934,Z 304.234,A -85,B 0,C 180,E1 -25145.172,E2 -25145.172} C_VEL
LIN {X 0,Y 128.903,Z 304.238,A -85,B 0,C 180,E1 -25150.864,E2 -25150.864} C_VEL
LIN {X 0,Y 128.894,Z 304.237,A -85,B 0,C 180,E1 -25155.141,E2 -25155.141} C_VEL
LIN {X 0,Y 128.92,Z 304.233,A -85,B 0,C 180,E1 -25159.748,E2 -25159.748} C_VEL
LIN {X 0,Y 128.944,Z 304.235,A -85,B 0,C 180,E1 -25164.843,E2 -25164.843} C_VEL
LIN {X 0,Y 129.006,Z 304.227,A -85,B 0,C 180,E1 -25170.652,E2 -25170.652} C_VEL
LIN {X 0,Y 129.144,Z 304.18,A -85,B 0,C 180,E1 -25177.691,E2 -25177.691} C_VEL
LIN {X 0,Y 130.781,Z 304.111,A -85,B 0,C 180,E1 -25186.909,E2 -25186.909} C_VEL
LIN {X 0,Y 131.918,Z 314.451,A -85,B 0,C 180,E1 -25187.902,E2 -25187.902} C_VEL
LIN {X 0,Y 132.18,Z 363.818,A -85,B 0,C 180,E1 -25193.523,E2 -25193.523} C_VEL
LIN {X 0,Y 132.053,Z 377.072,A -85,B 0,C 180,E1 -25195.336,E2 -25195.336} C_VEL
LIN {X 0,Y 131.771,Z 389.267,A -85,B 0,C 180,E1 -25197.717,E2 -25197.717} C_VEL
LIN {X 0,Y 131.541,Z 398.358,A -85,B 0,C 180,E1 -25200.01,E2 -25200.01} C_VEL
LIN {X 0,Y 131.413,Z 406.919,A -85,B 0,C 180,E1 -25202.692,E2 -25202.692} C_VEL
LIN {X 0,Y 131.121,Z 417.402,A -85,B 0,C 180,E1 -25206.936,E2 -25206.936} C_VEL
LIN {X 0,Y 131.466,Z 425.181,A -85,B 0,C 180,E1 -25210.793,E2 -25210.793} C_VEL
LIN {X 0,Y 132.324,Z 431.566,A -85,B 0,C 180,E1 -25214.622,E2 -25214.622} C_VEL
LIN {X 0,Y 134.473,Z 438.457,A -85,B 0,C 180,E1 -25219.334,E2 -25219.334} C_VEL
LIN {X 0,Y 138.142,Z 444.317,A -85,B 0,C 180,E1 -25224.026,E2 -25224.026} C_VEL
LIN {X 0,Y 142.66,Z 448.56,A -85,B 0,C 180,E1 -25227.914,E2 -25227.914} C_VEL
LIN {X 0,Y 147.979,Z 451.792,A -85,B 0,C 180,E1 -25231.504,E2 -25231.504} C_VEL
LIN {X 0,Y 152.75,Z 453.775,A -85,B 0,C 180,E1 -25234.087,E2 -25234.087} C_VEL
LIN {X 0,Y 161.095,Z 455.623,A -85,B 0,C 180,E1 -25237.654,E2 -25237.654} C_VEL
LIN {X 0,Y 166.06,Z 456.158,A -85,B 0,C 180,E1 -25239.416,E2 -25239.416} C_VEL
LIN {X 0,Y 171.246,Z 456.162,A -85,B 0,C 180,E1 -25241.053,E2 -25241.053} C_VEL
LIN {X 0,Y 180.078,Z 455.407,A -85,B 0,C 180,E1 -25243.389,E2 -25243.389} C_VEL
LIN {X 0,Y 180.406,Z 455.47,A -85,B 0,C 180,E1 -25244.028,E2 -25244.028} C_VEL
LIN {X 0,Y 172.217,Z 457.034,A -85,B 0,C 180,E1 -25246.071,E2 -25246.071} C_VEL
LIN {X 0,Y 166.839,Z 457.597,A -85,B 0,C 180,E1 -25247.623,E2 -25247.623} C_VEL
LIN {X 0,Y 157.003,Z 457.646,A -85,B 0,C 180,E1 -25251.193,E2 -25251.193} C_VEL
LIN {X 0,Y 148.528,Z 456.215,A -85,B 0,C 180,E1 -25255.401,E2 -25255.401} C_VEL
LIN {X 0,Y 144.796,Z 455.044,A -85,B 0,C 180,E1 -25257.729,E2 -25257.729} C_VEL
LIN {X 0,Y 141.434,Z 453.426,A -85,B 0,C 180,E1 -25260.204,E2 -25260.204} C_VEL
LIN {X 0,Y 136.42,Z 449.31,A -85,B 0,C 180,E1 -25265.66,E2 -25265.66} C_VEL
LIN {X 0,Y 133.944,Z 445.093,A -85,B 0,C 180,E1 -25270.218,E2 -25270.218} C_VEL
LIN {X 0,Y 132.881,Z 441.52,A -85,B 0,C 180,E1 -25273.636,E2 -25273.636} C_VEL
LIN {X 0,Y 130.857,Z 445.132,A -85,B 0,C 180,E1 -25275.553,E2 -25275.553} C_VEL
LIN {X 0,Y 128.675,Z 450.249,A -85,B 0,C 180,E1 -25278.979,E2 -25278.979} C_VEL
LIN {X 0,Y 127.521,Z 453.983,A -85,B 0,C 180,E1 -25282.08,E2 -25282.08} C_VEL
LIN {X 0,Y 126.913,Z 457.415,A -85,B 0,C 180,E1 -25285.745,E2 -25285.745} C_VEL
LIN {X 0,Y 126.465,Z 458.69,A -85,B 0,C 180,E1 -25287.424,E2 -25287.424} C_VEL
LIN {X 0,Y 124.959,Z 460.283,A -85,B 0,C 180,E1 -25289.944,E2 -25289.944} C_VEL
LIN {X 0,Y 121.725,Z 462.035,A -85,B 0,C 180,E1 -25294.267,E2 -25294.267} C_VEL
LIN {X 0,Y 120.027,Z 462.881,A -85,B 0,C 180,E1 -25297.962,E2 -25297.962} C_VEL
LIN {X 0,Y 119.978,Z 463.1,A -85,B 0,C 180,E1 -25299.862,E2 -25299.862} C_VEL
LIN {X 0,Y 120.815,Z 463.313,A -85,B 0,C 180,E1 -25303.455,E2 -25303.455} C_VEL
LIN {X 0,Y 121.988,Z 462.928,A -85,B 0,C 180,E1 -25306.741,E2 -25306.741} C_VEL
LIN {X 0,Y 123.574,Z 462.026,A -85,B 0,C 180,E1 -25309.952,E2 -25309.952} C_VEL
LIN {X 0,Y 125.573,Z 460.672,A -85,B 0,C 180,E1 -25313.064,E2 -25313.064} C_VEL
LIN {X 0,Y 129.391,Z 457.672,A -85,B 0,C 180,E1 -25317.495,E2 -25317.495} C_VEL
LIN {X 0,Y 132.415,Z 454.965,A -85,B 0,C 180,E1 -25320.279,E2 -25320.279} C_VEL
LIN {X 0,Y 135.65,Z 451.66,A -85,B 0,C 180,E1 -25322.956,E2 -25322.956} C_VEL
LIN {X 0,Y 140.274,Z 446.494,A -85,B 0,C 180,E1 -25326.064,E2 -25326.064} C_VEL
LIN {X 0,Y 144.179,Z 441.47,A -85,B 0,C 180,E1 -25328.425,E2 -25328.425} C_VEL
LIN {X 0,Y 148.552,Z 435.282,A -85,B 0,C 180,E1 -25330.657,E2 -25330.657} C_VEL
LIN {X 0,Y 152.619,Z 428.573,A -85,B 0,C 180,E1 -25332.58,E2 -25332.58} C_VEL
LIN {X 0,Y 156.385,Z 421.518,A -85,B 0,C 180,E1 -25334.152,E2 -25334.152} C_VEL
LIN {X 0,Y 160.01,Z 413.551,A -85,B 0,C 180,E1 -25335.539,E2 -25335.539} C_VEL
LIN {X 0,Y 163.211,Z 405.308,A -85,B 0,C 180,E1 -25336.606,E2 -25336.606} C_VEL
LIN {X 0,Y 166.174,Z 395.476,A -85,B 0,C 180,E1 -25337.574,E2 -25337.574} C_VEL
LIN {X 0,Y 168.605,Z 384.098,A -85,B 0,C 180,E1 -25338.361,E2 -25338.361} C_VEL
LIN {X 0,Y 169.646,Z 374.949,A -85,B 0,C 180,E1 -25338.807,E2 -25338.807} C_VEL
LIN {X 0,Y 166.154,Z 365.437,A -85,B 0,C 180,E1 -25341.39,E2 -25341.39} C_VEL
LIN {X 0,Y 162.457,Z 356.988,A -85,B 0,C 180,E1 -25344.395,E2 -25344.395} C_VEL
LIN {X 0,Y 158.56,Z 348.832,A -85,B 0,C 180,E1 -25348.016,E2 -25348.016} C_VEL
LIN {X 0,Y 155.656,Z 343.54,A -85,B 0,C 180,E1 -25351.125,E2 -25351.125} C_VEL
LIN {X 0,Y 153.272,Z 339.75,A -85,B 0,C 180,E1 -25354.066,E2 -25354.066} C_VEL
LIN {X 0,Y 150.991,Z 336.924,A -85,B 0,C 180,E1 -25357.41,E2 -25357.41} C_VEL
LIN {X 0,Y 150.175,Z 335.092,A -85,B 0,C 180,E1 -25359.034,E2 -25359.034} C_VEL
LIN {X 0,Y 147.363,Z 332.073,A -85,B 0,C 180,E1 -25366.541,E2 -25366.541} C_VEL
LIN {X 0,Y 146.991,Z 329.736,A -85,B 0,C 180,E1 -25371.051,E2 -25371.051} C_VEL
LIN {X 0,Y 147.072,Z 329.932,A -85,B 0,C 180,E1 -25374.06,E2 -25374.06} C_VEL
LIN {X 0,Y 147.642,Z 331.277,A -85,B 0,C 180,E1 -25377.815,E2 -25377.815} C_VEL
LIN {X 0,Y 149.526,Z 334.441,A -85,B 0,C 180,E1 -25383.359,E2 -25383.359} C_VEL
LIN {X 0,Y 150.549,Z 335.265,A -85,B 0,C 180,E1 -25385.264,E2 -25385.264} C_VEL
LIN {X 0,Y 152.586,Z 338.809,A -85,B 0,C 180,E1 -25388.69,E2 -25388.69} C_VEL
LIN {X 0,Y 153.85,Z 340.392,A -85,B 0,C 180,E1 -25390.338,E2 -25390.338} C_VEL
LIN {X 0,Y 157.047,Z 345.134,A -85,B 0,C 180,E1 -25393.992,E2 -25393.992} C_VEL
LIN {X 0,Y 160.065,Z 349.764,A -85,B 0,C 180,E1 -25396.902,E2 -25396.902} C_VEL
LIN {X 0,Y 163.749,Z 355.745,A -85,B 0,C 180,E1 -25399.991,E2 -25399.991} C_VEL
LIN {X 0,Y 168.234,Z 363.915,A -85,B 0,C 180,E1 -25403.299,E2 -25403.299} C_VEL
LIN {X 0,Y 170.183,Z 367.818,A -85,B 0,C 180,E1 -25404.636,E2 -25404.636} C_VEL
LIN {X 0,Y 168.761,Z 378.225,A -85,B 0,C 180,E1 -25405.198,E2 -25405.198} C_VEL
LIN {X 0,Y 166.939,Z 387.094,A -85,B 0,C 180,E1 -25405.926,E2 -25405.926} C_VEL
LIN {X 0,Y 164.505,Z 395.875,A -85,B 0,C 180,E1 -25406.898,E2 -25406.898} C_VEL
LIN {X 0,Y 161.424,Z 404.587,A -85,B 0,C 180,E1 -25408.161,E2 -25408.161} C_VEL
LIN {X 0,Y 158.051,Z 412.269,A -85,B 0,C 180,E1 -25409.565,E2 -25409.565} C_VEL
LIN {X 0,Y 153.675,Z 420.765,A -85,B 0,C 180,E1 -25411.596,E2 -25411.596} C_VEL
LIN {X 0,Y 148.797,Z 428.677,A -85,B 0,C 180,E1 -25414.118,E2 -25414.118} C_VEL
LIN {X 0,Y 144.395,Z 434.593,A -85,B 0,C 180,E1 -25416.575,E2 -25416.575} C_VEL
LIN {X 0,Y 140.434,Z 439.352,A -85,B 0,C 180,E1 -25419.133,E2 -25419.133} C_VEL
LIN {X 0,Y 136.478,Z 443.492,A -85,B 0,C 180,E1 -25422.009,E2 -25422.009} C_VEL
LIN {X 0,Y 131.802,Z 447.643,A -85,B 0,C 180,E1 -25426.117,E2 -25426.117} C_VEL
LIN {X 0,Y 128.049,Z 450.366,A -85,B 0,C 180,E1 -25430.191,E2 -25430.191} C_VEL
LIN {X 0,Y 126.437,Z 451.4,A -85,B 0,C 180,E1 -25432.308,E2 -25432.308} C_VEL
LIN {X 0,Y 124.272,Z 452.365,A -85,B 0,C 180,E1 -25435.561,E2 -25435.561} C_VEL
LIN {X 0,Y 122.235,Z 452.797,A -85,B 0,C 180,E1 -25439.567,E2 -25439.567} C_VEL
LIN {X 0,Y 120.113,Z 451.954,A -85,B 0,C 180,E1 -25445.822,E2 -25445.822} C_VEL
LIN {X 0,Y 119.408,Z 450.307,A -85,B 0,C 180,E1 -25450.304,E2 -25450.304} C_VEL
LIN {X 0,Y 119.277,Z 447.853,A -85,B 0,C 180,E1 -25454.625,E2 -25454.625} C_VEL
LIN {X 0,Y 119.739,Z 443.624,A -85,B 0,C 180,E1 -25459.859,E2 -25459.859} C_VEL
LIN {X 0,Y 120.971,Z 437.891,A -85,B 0,C 180,E1 -25465.001,E2 -25465.001} C_VEL
LIN {X 0,Y 122.318,Z 431.621,A -85,B 0,C 180,E1 -25469.178,E2 -25469.178} C_VEL
LIN {X 0,Y 123.763,Z 425.491,A -85,B 0,C 180,E1 -25472.442,E2 -25472.442} C_VEL
LIN {X 0,Y 125.566,Z 418.016,A -85,B 0,C 180,E1 -25475.622,E2 -25475.622} C_VEL
LIN {X 0,Y 127.273,Z 410.754,A -85,B 0,C 180,E1 -25478.095,E2 -25478.095} C_VEL
LIN {X 0,Y 128.901,Z 403.026,A -85,B 0,C 180,E1 -25480.216,E2 -25480.216} C_VEL
LIN {X 0,Y 130.484,Z 394.526,A -85,B 0,C 180,E1 -25482.049,E2 -25482.049} C_VEL
LIN {X 0,Y 131.774,Z 385.145,A -85,B 0,C 180,E1 -25483.612,E2 -25483.612} C_VEL
LIN {X 0,Y 133.067,Z 373.174,A -85,B 0,C 180,E1 -25484.97,E2 -25484.97} C_VEL
LIN {X 0,Y 134.007,Z 356.433,A -85,B 0,C 180,E1 -25485.954,E2 -25485.954} C_VEL
LIN {X 0,Y 135.1,Z 332.67,A -85,B 0,C 180,E1 -25487.148,E2 -25487.148} C_VEL
LIN {X 0,Y 128.657,Z 318.27,A -85,B 0,C 180,E1 -25489.567,E2 -25489.567} C_VEL
LIN {X 0,Y 123.478,Z 308.519,A -85,B 0,C 180,E1 -25491.619,E2 -25491.619} C_VEL
LIN {X 0,Y 122.195,Z 305.871,A -85,B 0,C 180,E1 -25492.177,E2 -25492.177} C_VEL
LIN {X 0,Y 122.06,Z 305.094,A -85,B 0,C 180,E1 -25492.283,E2 -25492.283} C_VEL
LIN {X 0,Y 121.915,Z 305.113,A -85,B 0,C 180,E1 -25497.464,E2 -25497.464} C_VEL
LIN {X 0,Y 121.875,Z 305.1,A -85,B 0,C 180,E1 -25501.265,E2 -25501.265} C_VEL
LIN {X 0,Y 121.859,Z 305.116,A -85,B 0,C 180,E1 -25506.176,E2 -25506.176} C_VEL
LIN {X 0,Y 121.844,Z 305.119,A -85,B 0,C 180,E1 -25511.441,E2 -25511.441} C_VEL
LIN {X 0,Y 121.848,Z 305.118,A -85,B 0,C 180,E1 -25518.576,E2 -25518.576} C_VEL
LIN {X 0,Y 121.896,Z 305.113,A -85,B 0,C 180,E1 -25524.806,E2 -25524.806} C_VEL
LIN {X 0,Y 121.915,Z 305.109,A -85,B 0,C 180,E1 -25529.85,E2 -25529.85} C_VEL
LIN {X 0,Y 122.079,Z 305.063,A -85,B 0,C 180,E1 -25537.091,E2 -25537.091} C_VEL
LIN {X 0,Y 124.048,Z 304.846,A -85,B 0,C 180,E1 -25547.848,E2 -25547.848} C_VEL
LIN {X 0,Y 125.162,Z 314.595,A -85,B 0,C 180,E1 -25548.882,E2 -25548.882} C_VEL
LIN {X 0,Y 125.701,Z 365.166,A -85,B 0,C 180,E1 -25554.999,E2 -25554.999} C_VEL
LIN {X 0,Y 125.571,Z 377.395,A -85,B 0,C 180,E1 -25556.802,E2 -25556.802} C_VEL
LIN {X 0,Y 125.428,Z 388.954,A -85,B 0,C 180,E1 -25559.208,E2 -25559.208} C_VEL
LIN {X 0,Y 125.235,Z 399.184,A -85,B 0,C 180,E1 -25562.02,E2 -25562.02} C_VEL
LIN {X 0,Y 125.089,Z 407.444,A -85,B 0,C 180,E1 -25564.845,E2 -25564.845} C_VEL
LIN {X 0,Y 124.939,Z 416.888,A -85,B 0,C 180,E1 -25568.909,E2 -25568.909} C_VEL
LIN {X 0,Y 125.494,Z 424.545,A -85,B 0,C 180,E1 -25572.955,E2 -25572.955} C_VEL
LIN {X 0,Y 126.913,Z 432.208,A -85,B 0,C 180,E1 -25577.742,E2 -25577.742} C_VEL
LIN {X 0,Y 130.094,Z 439.533,A -85,B 0,C 180,E1 -25583.014,E2 -25583.014} C_VEL
LIN {X 0,Y 134.913,Z 445.494,A -85,B 0,C 180,E1 -25587.968,E2 -25587.968} C_VEL
LIN {X 0,Y 140.149,Z 449.526,A -85,B 0,C 180,E1 -25591.782,E2 -25591.782} C_VEL
LIN {X 0,Y 147.386,Z 453.105,A -85,B 0,C 180,E1 -25595.841,E2 -25595.841} C_VEL
LIN {X 0,Y 150.692,Z 454.301,A -85,B 0,C 180,E1 -25597.331,E2 -25597.331} C_VEL
LIN {X 0,Y 160.61,Z 456.257,A -85,B 0,C 180,E1 -25601.033,E2 -25601.033} C_VEL
LIN {X 0,Y 168.622,Z 456.721,A -85,B 0,C 180,E1 -25603.408,E2 -25603.408} C_VEL
LIN {X 0,Y 168.297,Z 456.858,A -85,B 0,C 180,E1 -25604.076,E2 -25604.076} C_VEL
LIN {X 0,Y 161.658,Z 457.188,A -85,B 0,C 180,E1 -25605.925,E2 -25605.925} C_VEL
LIN {X 0,Y 156.458,Z 457.127,A -85,B 0,C 180,E1 -25607.639,E2 -25607.639} C_VEL
LIN {X 0,Y 147.073,Z 455.782,A -85,B 0,C 180,E1 -25611.594,E2 -25611.594} C_VEL
LIN {X 0,Y 142.891,Z 454.705,A -85,B 0,C 180,E1 -25613.827,E2 -25613.827} C_VEL
LIN {X 0,Y 135.604,Z 451.278,A -85,B 0,C 180,E1 -25618.783,E2 -25618.783} C_VEL
LIN {X 0,Y 131.527,Z 447.958,A -85,B 0,C 180,E1 -25622.986,E2 -25622.986} C_VEL
LIN {X 0,Y 128.698,Z 443.784,A -85,B 0,C 180,E1 -25627.526,E2 -25627.526} C_VEL
LIN {X 0,Y 127.075,Z 439.073,A -85,B 0,C 180,E1 -25632.001,E2 -25632.001} C_VEL
LIN {X 0,Y 124.063,Z 444.182,A -85,B 0,C 180,E1 -25634.744,E2 -25634.744} C_VEL
LIN {X 0,Y 121.778,Z 449.432,A -85,B 0,C 180,E1 -25638.346,E2 -25638.346} C_VEL
LIN {X 0,Y 120.161,Z 454.798,A -85,B 0,C 180,E1 -25643.282,E2 -25643.282} C_VEL
LIN {X 0,Y 119.789,Z 457.65,A -85,B 0,C 180,E1 -25646.636,E2 -25646.636} C_VEL
LIN {X 0,Y 119.854,Z 459.908,A -85,B 0,C 180,E1 -25649.999,E2 -25649.999} C_VEL
LIN {X 0,Y 119.61,Z 461.479,A -85,B 0,C 180,E1 -25653.368,E2 -25653.368} C_VEL
LIN {X 0,Y 119.643,Z 462.54,A -85,B 0,C 180,E1 -25656.746,E2 -25656.746} C_VEL
LIN {X 0,Y 119.978,Z 463.1,A -85,B 0,C 180,E1 -25659.862,E2 -25659.862} C_VEL
LIN {X 0,Y 119.906,Z 463.386,A -85,B 0,C 180,E1 -25662.684,E2 -25662.684} C_VEL
LIN {X 0,Y 118.626,Z 462.972,A -85,B 0,C 180,E1 -25667.413,E2 -25667.413} C_VEL
LIN {X 0,Y 118.206,Z 461.564,A -85,B 0,C 180,E1 -25672.166,E2 -25672.166} C_VEL
LIN {X 0,Y 119.444,Z 460.282,A -85,B 0,C 180,E1 -25674.886,E2 -25674.886} C_VEL
LIN {X 0,Y 123.142,Z 457.633,A -85,B 0,C 180,E1 -25679.019,E2 -25679.019} C_VEL
LIN {X 0,Y 126.328,Z 455.019,A -85,B 0,C 180,E1 -25681.904,E2 -25681.904} C_VEL
LIN {X 0,Y 131.631,Z 449.889,A -85,B 0,C 180,E1 -25685.965,E2 -25685.965} C_VEL
LIN {X 0,Y 136.653,Z 444.402,A -85,B 0,C 180,E1 -25689.05,E2 -25689.05} C_VEL
LIN {X 0,Y 142.666,Z 436.684,A -85,B 0,C 180,E1 -25692.226,E2 -25692.226} C_VEL
LIN {X 0,Y 147.651,Z 429.01,A -85,B 0,C 180,E1 -25694.498,E2 -25694.498} C_VEL
LIN {X 0,Y 152.022,Z 421.195,A -85,B 0,C 180,E1 -25696.248,E2 -25696.248} C_VEL
LIN {X 0,Y 155.791,Z 413.228,A -85,B 0,C 180,E1 -25697.621,E2 -25697.621} C_VEL
LIN {X 0,Y 159.111,Z 404.985,A -85,B 0,C 180,E1 -25698.667,E2 -25698.667} C_VEL
LIN {X 0,Y 161.852,Z 396.283,A -85,B 0,C 180,E1 -25699.53,E2 -25699.53} C_VEL
LIN {X 0,Y 164.129,Z 386.634,A -85,B 0,C 180,E1 -25700.216,E2 -25700.216} C_VEL
LIN {X 0,Y 165.443,Z 377.598,A -85,B 0,C 180,E1 -25700.703,E2 -25700.703} C_VEL
LIN {X 0,Y 162.633,Z 369.283,A -85,B 0,C 180,E1 -25703.151,E2 -25703.151} C_VEL
LIN {X 0,Y 159.401,Z 361.665,A -85,B 0,C 180,E1 -25706.037,E2 -25706.037} C_VEL
LIN {X 0,Y 156.074,Z 354.332,A -85,B 0,C 180,E1 -25709.437,E2 -25709.437} C_VEL
LIN {X 0,Y 153.376,Z 349.132,A -85,B 0,C 180,E1 -25712.617,E2 -25712.617} C_VEL
LIN {X 0,Y 151.719,Z 346.424,A -85,B 0,C 180,E1 -25714.831,E2 -25714.831} C_VEL
LIN {X 0,Y 149.508,Z 343.384,A -85,B 0,C 180,E1 -25718.379,E2 -25718.379} C_VEL
LIN {X 0,Y 148.891,Z 341.92,A -85,B 0,C 180,E1 -25719.715,E2 -25719.715} C_VEL
LIN {X 0,Y 146.247,Z 338.645,A -85,B 0,C 180,E1 -25727.835,E2 -25727.835} C_VEL
LIN {X 0,Y 146.09,Z 336.718,A -85,B 0,C 180,E1 -25731.693,E2 -25731.693} C_VEL
LIN {X 0,Y 146.299,Z 337.323,A -85,B 0,C 180,E1 -25735.219,E2 -25735.219} C_VEL
LIN {X 0,Y 146.82,Z 338.89,A -85,B 0,C 180,E1 -25738.304,E2 -25738.304} C_VEL
LIN {X 0,Y 148.625,Z 341.527,A -85,B 0,C 180,E1 -25743.38,E2 -25743.38} C_VEL
LIN {X 0,Y 149.301,Z 342.252,A -85,B 0,C 180,E1 -25744.716,E2 -25744.716} C_VEL
LIN {X 0,Y 151.358,Z 345.76,A -85,B 0,C 180,E1 -25748.303,E2 -25748.303} C_VEL
LIN {X 0,Y 152.357,Z 347.244,A -85,B 0,C 180,E1 -25749.707,E2 -25749.707} C_VEL
LIN {X 0,Y 155.217,Z 351.633,A -85,B 0,C 180,E1 -25753.159,E2 -25753.159} C_VEL
LIN {X 0,Y 157.959,Z 356.053,A -85,B 0,C 180,E1 -25755.971,E2 -25755.971} C_VEL
LIN {X 0,Y 161.491,Z 362.146,A -85,B 0,C 180,E1 -25759.123,E2 -25759.123} C_VEL
LIN {X 0,Y 165.148,Z 369.286,A -85,B 0,C 180,E1 -25762.099,E2 -25762.099} C_VEL
LIN {X 0,Y 165.962,Z 371.088,A -85,B 0,C 180,E1 -25762.769,E2 -25762.769} C_VEL
LIN {X 0,Y 164.373,Z 380.848,A -85,B 0,C 180,E1 -25763.338,E2 -25763.338} C_VEL
LIN {X 0,Y 161.901,Z 391.311,A -85,B 0,C 180,E1 -25764.275,E2 -25764.275} C_VEL
LIN {X 0,Y 158.029,Z 402.738,A -85,B 0,C 180,E1 -25765.767,E2 -25765.767} C_VEL
LIN {X 0,Y 154.368,Z 411.138,A -85,B 0,C 180,E1 -25767.232,E2 -25767.232} C_VEL
LIN {X 0,Y 150.506,Z 418.55,A -85,B 0,C 180,E1 -25768.891,E2 -25768.891} C_VEL
LIN {X 0,Y 146.905,Z 424.512,A -85,B 0,C 180,E1 -25770.557,E2 -25770.557} C_VEL
LIN {X 0,Y 142.313,Z 431.107,A -85,B 0,C 180,E1 -25772.91,E2 -25772.91} C_VEL
LIN {X 0,Y 137.921,Z 436.52,A -85,B 0,C 180,E1 -25775.383,E2 -25775.383} C_VEL
LIN {X 0,Y 133.81,Z 440.98,A -85,B 0,C 180,E1 -25778.017,E2 -25778.017} C_VEL
LIN {X 0,Y 129.978,Z 444.628,A -85,B 0,C 180,E1 -25780.801,E2 -25780.801} C_VEL
LIN {X 0,Y 124.88,Z 448.747,A -85,B 0,C 180,E1 -25785.294,E2 -25785.294} C_VEL
LIN {X 0,Y 120.587,Z 451.503,A -85,B 0,C 180,E1 -25790.127,E2 -25790.127} C_VEL
LIN {X 0,Y 118.177,Z 452.532,A -85,B 0,C 180,E1 -25793.509,E2 -25793.509} C_VEL
LIN {X 0,Y 115.534,Z 453.134,A -85,B 0,C 180,E1 -25798.364,E2 -25798.364} C_VEL
LIN {X 0,Y 113.368,Z 452.469,A -85,B 0,C 180,E1 -25804.282,E2 -25804.282} C_VEL
LIN {X 0,Y 112.368,Z 450.627,A -85,B 0,C 180,E1 -25809.707,E2 -25809.707} C_VEL
LIN {X 0,Y 112.196,Z 447.393,A -85,B 0,C 180,E1 -25815.49,E2 -25815.49} C_VEL
LIN {X 0,Y 112.85,Z 442.895,A -85,B 0,C 180,E1 -25821.044,E2 -25821.044} C_VEL
LIN {X 0,Y 113.988,Z 437.806,A -85,B 0,C 180,E1 -25825.616,E2 -25825.616} C_VEL
LIN {X 0,Y 115.418,Z 431.5,A -85,B 0,C 180,E1 -25830.001,E2 -25830.001} C_VEL
LIN {X 0,Y 116.982,Z 425.277,A -85,B 0,C 180,E1 -25833.445,E2 -25833.445} C_VEL
LIN {X 0,Y 118.657,Z 418.736,A -85,B 0,C 180,E1 -25836.377,E2 -25836.377} C_VEL
LIN {X 0,Y 120.324,Z 412.056,A -85,B 0,C 180,E1 -25838.82,E2 -25838.82} C_VEL
LIN {X 0,Y 122.234,Z 403.471,A -85,B 0,C 180,E1 -25841.326,E2 -25841.326} C_VEL
LIN {X 0,Y 123.819,Z 395.573,A -85,B 0,C 180,E1 -25843.124,E2 -25843.124} C_VEL
LIN {X 0,Y 125.204,Z 386.26,A -85,B 0,C 180,E1 -25844.778,E2 -25844.778} C_VEL
LIN {X 0,Y 126.391,Z 376.413,A -85,B 0,C 180,E1 -25846.016,E2 -25846.016} C_VEL
LIN {X 0,Y 127.284,Z 363.692,A -85,B 0,C 180,E1 -25846.986,E2 -25846.986} C_VEL
LIN {X 0,Y 128.7,Z 334.233,A -85,B 0,C 180,E1 -25848.53,E2 -25848.53} C_VEL
LIN {X 0,Y 122.834,Z 321.257,A -85,B 0,C 180,E1 -25850.927,E2 -25850.927} C_VEL
LIN {X 0,Y 118.416,Z 312.82,A -85,B 0,C 180,E1 -25852.837,E2 -25852.837} C_VEL
LIN {X 0,Y 116.512,Z 309.628,A -85,B 0,C 180,E1 -25853.686,E2 -25853.686} C_VEL
LIN {X 0,Y 115.125,Z 307.177,A -85,B 0,C 180,E1 -25854.337,E2 -25854.337} C_VEL
LIN {X 0,Y 114.884,Z 305.989,A -85,B 0,C 180,E1 -25854.593,E2 -25854.593} C_VEL
LIN {X 0,Y 114.832,Z 305.977,A -85,B 0,C 180,E1 -25861.062,E2 -25861.062} C_VEL
LIN {X 0,Y 114.753,Z 305.996,A -85,B 0,C 180,E1 -25867.767,E2 -25867.767} C_VEL
LIN {X 0,Y 114.759,Z 305.999,A -85,B 0,C 180,E1 -25872.721,E2 -25872.721} C_VEL
LIN {X 0,Y 114.77,Z 306.002,A -85,B 0,C 180,E1 -25877.672,E2 -25877.672} C_VEL
LIN {X 0,Y 114.771,Z 306,A -85,B 0,C 180,E1 -25882.756,E2 -25882.756} C_VEL
LIN {X 0,Y 114.843,Z 305.988,A -85,B 0,C 180,E1 -25888.955,E2 -25888.955} C_VEL
LIN {X 0,Y 115.007,Z 305.949,A -85,B 0,C 180,E1 -25896.442,E2 -25896.442} C_VEL
LIN {X 0,Y 117.427,Z 305.669,A -85,B 0,C 180,E1 -25909.014,E2 -25909.014} C_VEL
LIN {X 0,Y 118.412,Z 314.475,A -85,B 0,C 180,E1 -25909.971,E2 -25909.971} C_VEL
LIN {X 0,Y 119.315,Z 362.903,A -85,B 0,C 180,E1 -25916.211,E2 -25916.211} C_VEL
LIN {X 0,Y 119.317,Z 375.354,A -85,B 0,C 180,E1 -25918.112,E2 -25918.112} C_VEL
LIN {X 0,Y 119.196,Z 386.638,A -85,B 0,C 180,E1 -25920.433,E2 -25920.433} C_VEL
LIN {X 0,Y 119.07,Z 397.276,A -85,B 0,C 180,E1 -25923.395,E2 -25923.395} C_VEL
LIN {X 0,Y 119,Z 404.61,A -85,B 0,C 180,E1 -25925.943,E2 -25925.943} C_VEL
LIN {X 0,Y 118.924,Z 412.518,A -85,B 0,C 180,E1 -25929.364,E2 -25929.364} C_VEL
LIN {X 0,Y 119.394,Z 420.887,A -85,B 0,C 180,E1 -25933.629,E2 -25933.629} C_VEL
LIN {X 0,Y 120.774,Z 429.1,A -85,B 0,C 180,E1 -25938.677,E2 -25938.677} C_VEL
LIN {X 0,Y 123.45,Z 436.01,A -85,B 0,C 180,E1 -25943.496,E2 -25943.496} C_VEL
LIN {X 0,Y 127.716,Z 442.11,A -85,B 0,C 180,E1 -25948.301,E2 -25948.301} C_VEL
LIN {X 0,Y 132.421,Z 446.568,A -85,B 0,C 180,E1 -25952.065,E2 -25952.065} C_VEL
LIN {X 0,Y 138.338,Z 450.415,A -85,B 0,C 180,E1 -25955.759,E2 -25955.759} C_VEL
LIN {X 0,Y 145.144,Z 453.451,A -85,B 0,C 180,E1 -25959.021,E2 -25959.021} C_VEL
LIN {X 0,Y 150.097,Z 455.027,A -85,B 0,C 180,E1 -25960.969,E2 -25960.969} C_VEL
LIN {X 0,Y 157.388,Z 456.525,A -85,B 0,C 180,E1 -25963.402,E2 -25963.402} C_VEL
LIN {X 0,Y 156.639,Z 456.587,A -85,B 0,C 180,E1 -25964.119,E2 -25964.119} C_VEL
LIN {X 0,Y 146.365,Z 455.309,A -85,B 0,C 180,E1 -25967.759,E2 -25967.759} C_VEL
LIN {X 0,Y 141.719,Z 454.282,A -85,B 0,C 180,E1 -25969.857,E2 -25969.857} C_VEL
LIN {X 0,Y 133.499,Z 451.038,A -85,B 0,C 180,E1 -25974.613,E2 -25974.613} C_VEL
LIN {X 0,Y 128.415,Z 447.75,A -85,B 0,C 180,E1 -25978.672,E2 -25978.672} C_VEL
LIN {X 0,Y 124.638,Z 443.778,A -85,B 0,C 180,E1 -25983.185,E2 -25983.185} C_VEL
LIN {X 0,Y 122.196,Z 439.134,A -85,B 0,C 180,E1 -25987.865,E2 -25987.865} C_VEL
LIN {X 0,Y 121.285,Z 436.555,A -85,B 0,C 180,E1 -25990.335,E2 -25990.335} C_VEL
LIN {X 0,Y 117.296,Z 443.176,A -85,B 0,C 180,E1 -25993.843,E2 -25993.843} C_VEL
LIN {X 0,Y 114.901,Z 448.567,A -85,B 0,C 180,E1 -25997.638,E2 -25997.638} C_VEL
LIN {X 0,Y 113.14,Z 454.091,A -85,B 0,C 180,E1 -26002.863,E2 -26002.863} C_VEL
LIN {X 0,Y 112.726,Z 457.03,A -85,B 0,C 180,E1 -26006.425,E2 -26006.425} C_VEL
LIN {X 0,Y 112.775,Z 459.317,A -85,B 0,C 180,E1 -26009.999,E2 -26009.999} C_VEL
LIN {X 0,Y 112.531,Z 460.948,A -85,B 0,C 180,E1 -26013.58,E2 -26013.58} C_VEL
LIN {X 0,Y 112.59,Z 462.091,A -85,B 0,C 180,E1 -26017.171,E2 -26017.171} C_VEL
LIN {X 0,Y 113.037,Z 462.778,A -85,B 0,C 180,E1 -26020.749,E2 -26020.749} C_VEL
LIN {X 0,Y 113.916,Z 462.999,A -85,B 0,C 180,E1 -26024.286,E2 -26024.286} C_VEL
LIN {X 0,Y 115.194,Z 462.639,A -85,B 0,C 180,E1 -26027.76,E2 -26027.76} C_VEL
LIN {X 0,Y 116.901,Z 461.818,A -85,B 0,C 180,E1 -26031.144,E2 -26031.144} C_VEL
LIN {X 0,Y 119.444,Z 460.282,A -85,B 0,C 180,E1 -26034.886,E2 -26034.886} C_VEL
LIN {X 0,Y 120.953,Z 458.904,A -85,B 0,C 180,E1 -26037.514,E2 -26037.514} C_VEL
LIN {X 0,Y 122.26,Z 455.933,A -85,B 0,C 180,E1 -26041.94,E2 -26041.94} C_VEL
LIN {X 0,Y 124.198,Z 452.239,A -85,B 0,C 180,E1 -26046.114,E2 -26046.114} C_VEL
LIN {X 0,Y 126.593,Z 449.456,A -85,B 0,C 180,E1 -26048.25,E2 -26048.25} C_VEL
LIN {X 0,Y 132.311,Z 443.487,A -85,B 0,C 180,E1 -26051.602,E2 -26051.602} C_VEL
LIN {X 0,Y 138.194,Z 436.256,A -85,B 0,C 180,E1 -26054.508,E2 -26054.508} C_VEL
LIN {X 0,Y 143.37,Z 428.613,A -85,B 0,C 180,E1 -26056.765,E2 -26056.765} C_VEL
LIN {X 0,Y 147.874,Z 420.918,A -85,B 0,C 180,E1 -26058.464,E2 -26058.464} C_VEL
LIN {X 0,Y 151.798,Z 412.974,A -85,B 0,C 180,E1 -26059.81,E2 -26059.81} C_VEL
LIN {X 0,Y 155.351,Z 404.428,A -85,B 0,C 180,E1 -26060.872,E2 -26060.872} C_VEL
LIN {X 0,Y 158.159,Z 395.78,A -85,B 0,C 180,E1 -26061.703,E2 -26061.703} C_VEL
LIN {X 0,Y 160.373,Z 386.682,A -85,B 0,C 180,E1 -26062.345,E2 -26062.345} C_VEL
LIN {X 0,Y 161.432,Z 380.184,A -85,B 0,C 180,E1 -26062.732,E2 -26062.732} C_VEL
LIN {X 0,Y 159.185,Z 372.986,A -85,B 0,C 180,E1 -26065.062,E2 -26065.062} C_VEL
LIN {X 0,Y 156.53,Z 366.43,A -85,B 0,C 180,E1 -26067.693,E2 -26067.693} C_VEL
LIN {X 0,Y 153.633,Z 359.726,A -85,B 0,C 180,E1 -26070.965,E2 -26070.965} C_VEL
LIN {X 0,Y 151.548,Z 355.401,A -85,B 0,C 180,E1 -26073.669,E2 -26073.669} C_VEL
LIN {X 0,Y 150.203,Z 353.082,A -85,B 0,C 180,E1 -26075.601,E2 -26075.601} C_VEL
LIN {X 0,Y 148.089,Z 349.894,A -85,B 0,C 180,E1 -26079.322,E2 -26079.322} C_VEL
LIN {X 0,Y 147.57,Z 348.759,A -85,B 0,C 180,E1 -26080.518,E2 -26080.518} C_VEL
LIN {X 0,Y 145.256,Z 345.384,A -85,B 0,C 180,E1 -26088.652,E2 -26088.652} C_VEL
LIN {X 0,Y 145.201,Z 343.783,A -85,B 0,C 180,E1 -26091.642,E2 -26091.642} C_VEL
LIN {X 0,Y 145.435,Z 344.466,A -85,B 0,C 180,E1 -26095.445,E2 -26095.445} C_VEL
LIN {X 0,Y 147.399,Z 348.383,A -85,B 0,C 180,E1 -26102.724,E2 -26102.724} C_VEL
LIN {X 0,Y 148.032,Z 349.136,A -85,B 0,C 180,E1 -26104.075,E2 -26104.075} C_VEL
LIN {X 0,Y 150.238,Z 352.816,A -85,B 0,C 180,E1 -26108.058,E2 -26108.058} C_VEL
LIN {X 0,Y 153.279,Z 357.917,A -85,B 0,C 180,E1 -26112.142,E2 -26112.142} C_VEL
LIN {X 0,Y 156.741,Z 363.697,A -85,B 0,C 180,E1 -26115.848,E2 -26115.848} C_VEL
LIN {X 0,Y 160.701,Z 371.545,A -85,B 0,C 180,E1 -26119.636,E2 -26119.636} C_VEL
LIN {X 0,Y 161.9,Z 374.315,A -85,B 0,C 180,E1 -26120.752,E2 -26120.752} C_VEL
LIN {X 0,Y 159.83,Z 385.229,A -85,B 0,C 180,E1 -26121.539,E2 -26121.539} C_VEL
LIN {X 0,Y 157.338,Z 394.057,A -85,B 0,C 180,E1 -26122.406,E2 -26122.406} C_VEL
LIN {X 0,Y 153.6,Z 404.157,A -85,B 0,C 180,E1 -26123.781,E2 -26123.781} C_VEL
LIN {X 0,Y 149.705,Z 412.496,A -85,B 0,C 180,E1 -26125.257,E2 -26125.257} C_VEL
LIN {X 0,Y 145.137,Z 420.658,A -85,B 0,C 180,E1 -26127.156,E2 -26127.156} C_VEL
LIN {X 0,Y 139.617,Z 428.939,A -85,B 0,C 180,E1 -26129.736,E2 -26129.736} C_VEL
LIN {X 0,Y 133.716,Z 436.015,A -85,B 0,C 180,E1 -26132.76,E2 -26132.76} C_VEL
LIN {X 0,Y 129.348,Z 440.627,A -85,B 0,C 180,E1 -26135.413,E2 -26135.413} C_VEL
LIN {X 0,Y 125.223,Z 444.416,A -85,B 0,C 180,E1 -26138.212,E2 -26138.212} C_VEL
LIN {X 0,Y 121.431,Z 447.482,A -85,B 0,C 180,E1 -26141.203,E2 -26141.203} C_VEL
LIN {X 0,Y 117.994,Z 449.846,A -85,B 0,C 180,E1 -26144.378,E2 -26144.378} C_VEL
LIN {X 0,Y 114.911,Z 451.554,A -85,B 0,C 180,E1 -26147.72,E2 -26147.72} C_VEL
LIN {X 0,Y 112.233,Z 452.699,A -85,B 0,C 180,E1 -26151.231,E2 -26151.231} C_VEL
LIN {X 0,Y 108.889,Z 453.471,A -85,B 0,C 180,E1 -26157.015,E2 -26157.015} C_VEL
LIN {X 0,Y 106.689,Z 452.975,A -85,B 0,C 180,E1 -26162.542,E2 -26162.542} C_VEL
LIN {X 0,Y 105.338,Z 450.943,A -85,B 0,C 180,E1 -26169.037,E2 -26169.037} C_VEL
LIN {X 0,Y 105.071,Z 448.145,A -85,B 0,C 180,E1 -26174.482,E2 -26174.482} C_VEL
LIN {X 0,Y 105.326,Z 445.382,A -85,B 0,C 180,E1 -26178.453,E2 -26178.453} C_VEL
LIN {X 0,Y 106.147,Z 441.157,A -85,B 0,C 180,E1 -26183.168,E2 -26183.168} C_VEL
LIN {X 0,Y 107.557,Z 435.399,A -85,B 0,C 180,E1 -26188.128,E2 -26188.128} C_VEL
LIN {X 0,Y 109.331,Z 428.466,A -85,B 0,C 180,E1 -26192.764,E2 -26192.764} C_VEL
LIN {X 0,Y 111.771,Z 419.457,A -85,B 0,C 180,E1 -26197.225,E2 -26197.225} C_VEL
LIN {X 0,Y 113.823,Z 411.606,A -85,B 0,C 180,E1 -26200.226,E2 -26200.226} C_VEL
LIN {X 0,Y 115.467,Z 404.618,A -85,B 0,C 180,E1 -26202.376,E2 -26202.376} C_VEL
LIN {X 0,Y 117.201,Z 396.615,A -85,B 0,C 180,E1 -26204.322,E2 -26204.322} C_VEL
LIN {X 0,Y 118.573,Z 388.348,A -85,B 0,C 180,E1 -26205.911,E2 -26205.911} C_VEL
LIN {X 0,Y 119.753,Z 378.943,A -85,B 0,C 180,E1 -26207.25,E2 -26207.25} C_VEL
LIN {X 0,Y 120.666,Z 369.384,A -85,B 0,C 180,E1 -26208.139,E2 -26208.139} C_VEL
LIN {X 0,Y 122.451,Z 336.147,A -85,B 0,C 180,E1 -26210.014,E2 -26210.014} C_VEL
LIN {X 0,Y 116.978,Z 324.006,A -85,B 0,C 180,E1 -26212.473,E2 -26212.473} C_VEL
LIN {X 0,Y 112.014,Z 314.642,A -85,B 0,C 180,E1 -26214.847,E2 -26214.847} C_VEL
LIN {X 0,Y 109.514,Z 310.708,A -85,B 0,C 180,E1 -26216.077,E2 -26216.077} C_VEL
LIN {X 0,Y 108.052,Z 308.265,A -85,B 0,C 180,E1 -26216.845,E2 -26216.845} C_VEL
LIN {X 0,Y 107.727,Z 306.879,A -85,B 0,C 180,E1 -26217.173,E2 -26217.173} C_VEL
LIN {X 0,Y 107.756,Z 306.857,A -85,B 0,C 180,E1 -26222.044,E2 -26222.044} C_VEL
LIN {X 0,Y 107.662,Z 306.878,A -85,B 0,C 180,E1 -26228.454,E2 -26228.454} C_VEL
LIN {X 0,Y 107.653,Z 306.885,A -85,B 0,C 180,E1 -26235.901,E2 -26235.901} C_VEL
LIN {X 0,Y 107.669,Z 306.879,A -85,B 0,C 180,E1 -26241.564,E2 -26241.564} C_VEL
LIN {X 0,Y 107.779,Z 306.866,A -85,B 0,C 180,E1 -26248.572,E2 -26248.572} C_VEL
LIN {X 0,Y 107.975,Z 306.817,A -85,B 0,C 180,E1 -26257.026,E2 -26257.026} C_VEL
LIN {X 0,Y 110.776,Z 306.494,A -85,B 0,C 180,E1 -26270.195,E2 -26270.195} C_VEL
LIN {X 0,Y 110.937,Z 306.733,A -85,B 0,C 180,E1 -26270.382,E2 -26270.382} C_VEL
LIN {X 0,Y 111.796,Z 313.943,A -85,B 0,C 180,E1 -26271.198,E2 -26271.198} C_VEL
LIN {X 0,Y 113.073,Z 362.602,A -85,B 0,C 180,E1 -26277.897,E2 -26277.897} C_VEL
LIN {X 0,Y 113.156,Z 375.089,A -85,B 0,C 180,E1 -26279.9,E2 -26279.9} C_VEL
LIN {X 0,Y 113.095,Z 385.813,A -85,B 0,C 180,E1 -26282.237,E2 -26282.237} C_VEL
LIN {X 0,Y 113.098,Z 396.95,A -85,B 0,C 180,E1 -26285.538,E2 -26285.538} C_VEL
LIN {X 0,Y 113.041,Z 405.766,A -85,B 0,C 180,E1 -26288.953,E2 -26288.953} C_VEL
LIN {X 0,Y 113.172,Z 413.445,A -85,B 0,C 180,E1 -26292.565,E2 -26292.565} C_VEL
LIN {X 0,Y 114.013,Z 421.383,A -85,B 0,C 180,E1 -26297.037,E2 -26297.037} C_VEL
LIN {X 0,Y 116.434,Z 430.686,A -85,B 0,C 180,E1 -26303.112,E2 -26303.112} C_VEL
LIN {X 0,Y 120.919,Z 438.44,A -85,B 0,C 180,E1 -26308.878,E2 -26308.878} C_VEL
LIN {X 0,Y 124.844,Z 442.844,A -85,B 0,C 180,E1 -26312.343,E2 -26312.343} C_VEL
LIN {X 0,Y 130.653,Z 447.478,A -85,B 0,C 180,E1 -26316.289,E2 -26316.289} C_VEL
LIN {X 0,Y 136.008,Z 450.64,A -85,B 0,C 180,E1 -26319.185,E2 -26319.185} C_VEL
LIN {X 0,Y 144.821,Z 454.178,A -85,B 0,C 180,E1 -26322.807,E2 -26322.807} C_VEL
LIN {X 0,Y 146.412,Z 454.799,A -85,B 0,C 180,E1 -26323.943,E2 -26323.943} C_VEL
LIN {X 0,Y 141.313,Z 453.763,A -85,B 0,C 180,E1 -26325.871,E2 -26325.871} C_VEL
LIN {X 0,Y 132.153,Z 450.695,A -85,B 0,C 180,E1 -26330.344,E2 -26330.344} C_VEL
LIN {X 0,Y 124.486,Z 446.21,A -85,B 0,C 180,E1 -26335.627,E2 -26335.627} C_VEL
LIN {X 0,Y 120.169,Z 442.104,A -85,B 0,C 180,E1 -26340.19,E2 -26340.19} C_VEL
LIN {X 0,Y 116.744,Z 436.31,A -85,B 0,C 180,E1 -26346.097,E2 -26346.097} C_VEL
LIN {X 0,Y 115.829,Z 433.79,A -85,B 0,C 180,E1 -26348.441,E2 -26348.441} C_VEL
LIN {X 0,Y 112.51,Z 438.832,A -85,B 0,C 180,E1 -26350.855,E2 -26350.855} C_VEL
LIN {X 0,Y 109.659,Z 444.035,A -85,B 0,C 180,E1 -26354.052,E2 -26354.052} C_VEL
LIN {X 0,Y 107.239,Z 449.724,A -85,B 0,C 180,E1 -26358.661,E2 -26358.661} C_VEL
LIN {X 0,Y 106.122,Z 453.382,A -85,B 0,C 180,E1 -26362.388,E2 -26362.388} C_VEL
LIN {X 0,Y 105.64,Z 457.562,A -85,B 0,C 180,E1 -26368.093,E2 -26368.093} C_VEL
LIN {X 0,Y 105.695,Z 458.702,A -85,B 0,C 180,E1 -26369.999,E2 -26369.999} C_VEL
LIN {X 0,Y 105.461,Z 460.417,A -85,B 0,C 180,E1 -26373.82,E2 -26373.82} C_VEL
LIN {X 0,Y 105.563,Z 461.642,A -85,B 0,C 180,E1 -26377.651,E2 -26377.651} C_VEL
LIN {X 0,Y 106.052,Z 462.408,A -85,B 0,C 180,E1 -26381.466,E2 -26381.466} C_VEL
LIN {X 0,Y 107.038,Z 462.654,A -85,B 0,C 180,E1 -26385.226,E2 -26385.226} C_VEL
LIN {X 0,Y 108.447,Z 462.351,A -85,B 0,C 180,E1 -26388.906,E2 -26388.906} C_VEL
LIN {X 0,Y 110.286,Z 461.61,A -85,B 0,C 180,E1 -26392.479,E2 -26392.479} C_VEL
LIN {X 0,Y 112.85,Z 460.288,A -85,B 0,C 180,E1 -26396.16,E2 -26396.16} C_VEL
LIN {X 0,Y 116.991,Z 457.595,A -85,B 0,C 180,E1 -26400.704,E2 -26400.704} C_VEL
LIN {X 0,Y 122.092,Z 453.54,A -85,B 0,C 180,E1 -26405.143,E2 -26405.143} C_VEL
LIN {X 0,Y 126.593,Z 449.456,A -85,B 0,C 180,E1 -26408.25,E2 -26408.25} C_VEL
LIN {X 0,Y 128.075,Z 447.566,A -85,B 0,C 180,E1 -26409.676,E2 -26409.676} C_VEL
LIN {X 0,Y 129.023,Z 444.358,A -85,B 0,C 180,E1 -26412.311,E2 -26412.311} C_VEL
LIN {X 0,Y 130.12,Z 440.935,A -85,B 0,C 180,E1 -26414.831,E2 -26414.831} C_VEL
LIN {X 0,Y 131.755,Z 438.478,A -85,B 0,C 180,E1 -26416.021,E2 -26416.021} C_VEL
LIN {X 0,Y 138.054,Z 430.26,A -85,B 0,C 180,E1 -26418.666,E2 -26418.666} C_VEL
LIN {X 0,Y 143.958,Z 420.691,A -85,B 0,C 180,E1 -26420.806,E2 -26420.806} C_VEL
LIN {X 0,Y 148.045,Z 412.765,A -85,B 0,C 180,E1 -26422.112,E2 -26422.112} C_VEL
LIN {X 0,Y 151.563,Z 404.613,A -85,B 0,C 180,E1 -26423.11,E2 -26423.11} C_VEL
LIN {X 0,Y 154.291,Z 396.689,A -85,B 0,C 180,E1 -26423.872,E2 -26423.872} C_VEL
LIN {X 0,Y 156.679,Z 387.594,A -85,B 0,C 180,E1 -26424.518,E2 -26424.518} C_VEL
LIN {X 0,Y 157.61,Z 382.787,A -85,B 0,C 180,E1 -26424.856,E2 -26424.856} C_VEL
LIN {X 0,Y 155.411,Z 375.548,A -85,B 0,C 180,E1 -26427.511,E2 -26427.511} C_VEL
LIN {X 0,Y 152.68,Z 368.42,A -85,B 0,C 180,E1 -26430.754,E2 -26430.754} C_VEL
LIN {X 0,Y 150.8,Z 363.9,A -85,B 0,C 180,E1 -26433.249,E2 -26433.249} C_VEL
LIN {X 0,Y 148.922,Z 359.946,A -85,B 0,C 180,E1 -26436.102,E2 -26436.102} C_VEL
LIN {X 0,Y 146.736,Z 356.469,A -85,B 0,C 180,E1 -26440.22,E2 -26440.22} C_VEL
LIN {X 0,Y 146.245,Z 355.509,A -85,B 0,C 180,E1 -26441.427,E2 -26441.427} C_VEL
LIN {X 0,Y 144.274,Z 352,A -85,B 0,C 180,E1 -26449.819,E2 -26449.819} C_VEL
LIN {X 0,Y 144.291,Z 351.008,A -85,B 0,C 180,E1 -26451.589,E2 -26451.589} C_VEL
LIN {X 0,Y 144.335,Z 350.914,A -85,B 0,C 180,E1 -26453.034,E2 -26453.034} C_VEL
LIN {X 0,Y 144.658,Z 352.148,A -85,B 0,C 180,E1 -26456.441,E2 -26456.441} C_VEL
LIN {X 0,Y 146.342,Z 355.353,A -85,B 0,C 180,E1 -26462.399,E2 -26462.399} C_VEL
LIN {X 0,Y 146.868,Z 356.139,A -85,B 0,C 180,E1 -26463.609,E2 -26463.609} C_VEL
LIN {X 0,Y 149.084,Z 360.138,A -85,B 0,C 180,E1 -26467.808,E2 -26467.808} C_VEL
LIN {X 0,Y 151.609,Z 364.592,A -85,B 0,C 180,E1 -26471.377,E2 -26471.377} C_VEL
LIN {X 0,Y 154.256,Z 369.353,A -85,B 0,C 180,E1 -26474.503,E2 -26474.503} C_VEL
LIN {X 0,Y 157.348,Z 376.047,A -85,B 0,C 180,E1 -26477.958,E2 -26477.958} C_VEL
LIN {X 0,Y 157.915,Z 378.012,A -85,B 0,C 180,E1 -26478.765,E2 -26478.765} C_VEL
LIN {X 0,Y 155.496,Z 388.469,A -85,B 0,C 180,E1 -26479.572,E2 -26479.572} C_VEL
LIN {X 0,Y 152.696,Z 397.302,A -85,B 0,C 180,E1 -26480.518,E2 -26480.518} C_VEL
LIN {X 0,Y 149.113,Z 406.166,A -85,B 0,C 180,E1 -26481.775,E2 -26481.775} C_VEL
LIN {X 0,Y 144.562,Z 415.156,A -85,B 0,C 180,E1 -26483.42,E2 -26483.42} C_VEL
LIN {X 0,Y 138.618,Z 424.601,A -85,B 0,C 180,E1 -26485.852,E2 -26485.852} C_VEL
LIN {X 0,Y 133.278,Z 431.611,A -85,B 0,C 180,E1 -26488.32,E2 -26488.32} C_VEL
LIN {X 0,Y 127.464,Z 437.986,A -85,B 0,C 180,E1 -26491.283,E2 -26491.283} C_VEL
LIN {X 0,Y 122.92,Z 442.29,A -85,B 0,C 180,E1 -26494,E2 -26494} C_VEL
LIN {X 0,Y 118.437,Z 445.955,A -85,B 0,C 180,E1 -26497.054,E2 -26497.054} C_VEL
LIN {X 0,Y 114.711,Z 448.606,A -85,B 0,C 180,E1 -26500.019,E2 -26500.019} C_VEL
LIN {X 0,Y 109.493,Z 451.607,A -85,B 0,C 180,E1 -26505.086,E2 -26505.086} C_VEL
LIN {X 0,Y 106.483,Z 452.869,A -85,B 0,C 180,E1 -26508.7,E2 -26508.7} C_VEL
LIN {X 0,Y 102.3,Z 453.809,A -85,B 0,C 180,E1 -26515.502,E2 -26515.502} C_VEL
LIN {X 0,Y 100.123,Z 453.42,A -85,B 0,C 180,E1 -26520.571,E2 -26520.571} C_VEL
LIN {X 0,Y 98.942,Z 452.447,A -85,B 0,C 180,E1 -26524.775,E2 -26524.775} C_VEL
LIN {X 0,Y 98.051,Z 450.07,A -85,B 0,C 180,E1 -26531.184,E2 -26531.184} C_VEL
LIN {X 0,Y 98.153,Z 446.261,A -85,B 0,C 180,E1 -26537.597,E2 -26537.597} C_VEL
LIN {X 0,Y 99.037,Z 441.54,A -85,B 0,C 180,E1 -26543.328,E2 -26543.328} C_VEL
LIN {X 0,Y 100.316,Z 436.559,A -85,B 0,C 180,E1 -26547.993,E2 -26547.993} C_VEL
LIN {X 0,Y 101.73,Z 431.251,A -85,B 0,C 180,E1 -26551.98,E2 -26551.98} C_VEL
LIN {X 0,Y 103.552,Z 424.849,A -85,B 0,C 180,E1 -26555.844,E2 -26555.844} C_VEL
LIN {X 0,Y 105.777,Z 417.057,A -85,B 0,C 180,E1 -26559.562,E2 -26559.562} C_VEL
LIN {X 0,Y 108.531,Z 406.752,A -85,B 0,C 180,E1 -26563.271,E2 -26563.271} C_VEL
LIN {X 0,Y 110.631,Z 397.661,A -85,B 0,C 180,E1 -26565.664,E2 -26565.664} C_VEL
LIN {X 0,Y 112.292,Z 388.374,A -85,B 0,C 180,E1 -26567.53,E2 -26567.53} C_VEL
LIN {X 0,Y 113.488,Z 379.369,A -85,B 0,C 180,E1 -26568.866,E2 -26568.866} C_VEL
LIN {X 0,Y 114.453,Z 370.108,A -85,B 0,C 180,E1 -26569.766,E2 -26569.766} C_VEL
LIN {X 0,Y 116.244,Z 338.054,A -85,B 0,C 180,E1 -26571.672,E2 -26571.672} C_VEL
LIN {X 0,Y 111.626,Z 327.66,A -85,B 0,C 180,E1 -26573.966,E2 -26573.966} C_VEL
LIN {X 0,Y 107.416,Z 319.445,A -85,B 0,C 180,E1 -26576.165,E2 -26576.165} C_VEL
LIN {X 0,Y 102.629,Z 311.852,A -85,B 0,C 180,E1 -26578.808,E2 -26578.808} C_VEL
LIN {X 0,Y 101.031,Z 309.353,A -85,B 0,C 180,E1 -26579.764,E2 -26579.764} C_VEL
LIN {X 0,Y 100.663,Z 307.744,A -85,B 0,C 180,E1 -26580.123,E2 -26580.123} C_VEL
LIN {X 0,Y 100.64,Z 307.752,A -85,B 0,C 180,E1 -26583.964,E2 -26583.964} C_VEL
LIN {X 0,Y 100.614,Z 307.759,A -85,B 0,C 180,E1 -26589.816,E2 -26589.816} C_VEL
LIN {X 0,Y 100.624,Z 307.759,A -85,B 0,C 180,E1 -26595.718,E2 -26595.718} C_VEL
LIN {X 0,Y 100.607,Z 307.757,A -85,B 0,C 180,E1 -26601.064,E2 -26601.064} C_VEL
LIN {X 0,Y 100.676,Z 307.75,A -85,B 0,C 180,E1 -26606.9,E2 -26606.9} C_VEL
LIN {X 0,Y 100.802,Z 307.725,A -85,B 0,C 180,E1 -26615.286,E2 -26615.286} C_VEL
LIN {X 0,Y 101.785,Z 307.615,A -85,B 0,C 180,E1 -26625.167,E2 -26625.167} C_VEL
LIN {X 0,Y 104.366,Z 307.288,A -85,B 0,C 180,E1 -26631.786,E2 -26631.786} C_VEL
LIN {X 0,Y 104.477,Z 307.274,A -85,B 0,C 180,E1 -26631.916,E2 -26631.916} C_VEL
LIN {X 0,Y 105.284,Z 314.098,A -85,B 0,C 180,E1 -26632.738,E2 -26632.738} C_VEL
LIN {X 0,Y 106.962,Z 361.365,A -85,B 0,C 180,E1 -26639.659,E2 -26639.659} C_VEL
LIN {X 0,Y 107.166,Z 374.359,A -85,B 0,C 180,E1 -26641.891,E2 -26641.891} C_VEL
LIN {X 0,Y 107.228,Z 384.571,A -85,B 0,C 180,E1 -26644.245,E2 -26644.245} C_VEL
LIN {X 0,Y 107.302,Z 395.457,A -85,B 0,C 180,E1 -26647.539,E2 -26647.539} C_VEL
LIN {X 0,Y 107.292,Z 404.698,A -85,B 0,C 180,E1 -26651.345,E2 -26651.345} C_VEL
LIN {X 0,Y 107.878,Z 414.003,A -85,B 0,C 180,E1 -26656.086,E2 -26656.086} C_VEL
LIN {X 0,Y 109.389,Z 423.165,A -85,B 0,C 180,E1 -26661.692,E2 -26661.692} C_VEL
LIN {X 0,Y 112.995,Z 432.006,A -85,B 0,C 180,E1 -26667.818,E2 -26667.818} C_VEL
LIN {X 0,Y 117.475,Z 438.36,A -85,B 0,C 180,E1 -26672.589,E2 -26672.589} C_VEL
LIN {X 0,Y 123.161,Z 443.824,A -85,B 0,C 180,E1 -26676.822,E2 -26676.822} C_VEL
LIN {X 0,Y 129.671,Z 448.308,A -85,B 0,C 180,E1 -26680.582,E2 -26680.582} C_VEL
LIN {X 0,Y 134.537,Z 450.902,A -85,B 0,C 180,E1 -26682.784,E2 -26682.784} C_VEL
LIN {X 0,Y 136.504,Z 451.818,A -85,B 0,C 180,E1 -26683.878,E2 -26683.878} C_VEL
LIN {X 0,Y 131.633,Z 450.206,A -85,B 0,C 180,E1 -26686.045,E2 -26686.045} C_VEL
LIN {X 0,Y 122.939,Z 445.907,A -85,B 0,C 180,E1 -26691.035,E2 -26691.035} C_VEL
LIN {X 0,Y 117.598,Z 441.825,A -85,B 0,C 180,E1 -26695.406,E2 -26695.406} C_VEL
LIN {X 0,Y 113.601,Z 437.138,A -85,B 0,C 180,E1 -26700.334,E2 -26700.334} C_VEL
LIN {X 0,Y 110.689,Z 430.828,A -85,B 0,C 180,E1 -26706.343,E2 -26706.343} C_VEL
LIN {X 0,Y 106.882,Z 436.192,A -85,B 0,C 180,E1 -26708.797,E2 -26708.797} C_VEL
LIN {X 0,Y 102.894,Z 443.14,A -85,B 0,C 180,E1 -26713.025,E2 -26713.025} C_VEL
LIN {X 0,Y 100.339,Z 448.92,A -85,B 0,C 180,E1 -26717.869,E2 -26717.869} C_VEL
LIN {X 0,Y 99.138,Z 452.658,A -85,B 0,C 180,E1 -26721.848,E2 -26721.848} C_VEL
LIN {X 0,Y 98.563,Z 456.831,A -85,B 0,C 180,E1 -26727.752,E2 -26727.752} C_VEL
LIN {X 0,Y 98.473,Z 459.115,A -85,B 0,C 180,E1 -26732.042,E2 -26732.042} C_VEL
LIN {X 0,Y 98.525,Z 461.193,A -85,B 0,C 180,E1 -26738.201,E2 -26738.201} C_VEL
LIN {X 0,Y 99.099,Z 462.027,A -85,B 0,C 180,E1 -26742.283,E2 -26742.283} C_VEL
LIN {X 0,Y 100.186,Z 462.285,A -85,B 0,C 180,E1 -26746.295,E2 -26746.295} C_VEL
LIN {X 0,Y 101.754,Z 462.064,A -85,B 0,C 180,E1 -26750.202,E2 -26750.202} C_VEL
LIN {X 0,Y 103.741,Z 461.403,A -85,B 0,C 180,E1 -26753.983,E2 -26753.983} C_VEL
LIN {X 0,Y 106.303,Z 460.298,A -85,B 0,C 180,E1 -26757.567,E2 -26757.567} C_VEL
LIN {X 0,Y 110.954,Z 457.56,A -85,B 0,C 180,E1 -26762.574,E2 -26762.574} C_VEL
LIN {X 0,Y 116.361,Z 453.608,A -85,B 0,C 180,E1 -26767.155,E2 -26767.155} C_VEL
LIN {X 0,Y 121.032,Z 449.711,A -85,B 0,C 180,E1 -26770.27,E2 -26770.27} C_VEL
LIN {X 0,Y 125.987,Z 444.963,A -85,B 0,C 180,E1 -26773.105,E2 -26773.105} C_VEL
LIN {X 0,Y 130.652,Z 439.753,A -85,B 0,C 180,E1 -26775.527,E2 -26775.527} C_VEL
LIN {X 0,Y 131.755,Z 438.478,A -85,B 0,C 180,E1 -26776.021,E2 -26776.021} C_VEL
LIN {X 0,Y 134.47,Z 434.684,A -85,B 0,C 180,E1 -26777.58,E2 -26777.58} C_VEL
LIN {X 0,Y 137.551,Z 428.073,A -85,B 0,C 180,E1 -26780.41,E2 -26780.41} C_VEL
LIN {X 0,Y 140.445,Z 420.922,A -85,B 0,C 180,E1 -26782.949,E2 -26782.949} C_VEL
LIN {X 0,Y 142.759,Z 416.132,A -85,B 0,C 180,E1 -26784.025,E2 -26784.025} C_VEL
LIN {X 0,Y 147.586,Z 405.905,A -85,B 0,C 180,E1 -26785.346,E2 -26785.346} C_VEL
LIN {X 0,Y 150.631,Z 397.676,A -85,B 0,C 180,E1 -26786.144,E2 -26786.144} C_VEL
LIN {X 0,Y 153.446,Z 387.512,A -85,B 0,C 180,E1 -26786.846,E2 -26786.846} C_VEL
LIN {X 0,Y 153.78,Z 385.592,A -85,B 0,C 180,E1 -26787.025,E2 -26787.025} C_VEL
LIN {X 0,Y 152.063,Z 378.897,A -85,B 0,C 180,E1 -26789.772,E2 -26789.772} C_VEL
LIN {X 0,Y 149.714,Z 371.921,A -85,B 0,C 180,E1 -26793.264,E2 -26793.264} C_VEL
LIN {X 0,Y 147.828,Z 367.458,A -85,B 0,C 180,E1 -26796.249,E2 -26796.249} C_VEL
LIN {X 0,Y 146.917,Z 365.907,A -85,B 0,C 180,E1 -26797.861,E2 -26797.861} C_VEL
LIN {X 0,Y 145.094,Z 362.392,A -85,B 0,C 180,E1 -26802.005,E2 -26802.005} C_VEL
LIN {X 0,Y 143.355,Z 358.853,A -85,B 0,C 180,E1 -26810.466,E2 -26810.466} C_VEL
LIN {X 0,Y 143.381,Z 358.243,A -85,B 0,C 180,E1 -26811.535,E2 -26811.535} C_VEL
LIN {X 0,Y 143.557,Z 358.479,A -85,B 0,C 180,E1 -26814.75,E2 -26814.75} C_VEL
LIN {X 0,Y 145.291,Z 362.315,A -85,B 0,C 180,E1 -26822.07,E2 -26822.07} C_VEL
LIN {X 0,Y 147.554,Z 366.66,A -85,B 0,C 180,E1 -26826.885,E2 -26826.885} C_VEL
LIN {X 0,Y 149.74,Z 370.988,A -85,B 0,C 180,E1 -26830.438,E2 -26830.438} C_VEL
LIN {X 0,Y 152.173,Z 375.986,A -85,B 0,C 180,E1 -26833.767,E2 -26833.767} C_VEL
LIN {X 0,Y 154.06,Z 381.153,A -85,B 0,C 180,E1 -26836.592,E2 -26836.592} C_VEL
LIN {X 0,Y 151.837,Z 390.033,A -85,B 0,C 180,E1 -26837.343,E2 -26837.343} C_VEL
LIN {X 0,Y 148.23,Z 400.545,A -85,B 0,C 180,E1 -26838.514,E2 -26838.514} C_VEL
LIN {X 0,Y 143.693,Z 410.358,A -85,B 0,C 180,E1 -26840.011,E2 -26840.011} C_VEL
LIN {X 0,Y 138.961,Z 418.531,A -85,B 0,C 180,E1 -26841.671,E2 -26841.671} C_VEL
LIN {X 0,Y 134.175,Z 425.545,A -85,B 0,C 180,E1 -26843.562,E2 -26843.562} C_VEL
LIN {X 0,Y 129.047,Z 431.951,A -85,B 0,C 180,E1 -26845.817,E2 -26845.817} C_VEL
LIN {X 0,Y 123.742,Z 437.519,A -85,B 0,C 180,E1 -26848.319,E2 -26848.319} C_VEL
LIN {X 0,Y 118.894,Z 441.973,A -85,B 0,C 180,E1 -26851.007,E2 -26851.007} C_VEL
LIN {X 0,Y 113.705,Z 446.055,A -85,B 0,C 180,E1 -26854.334,E2 -26854.334} C_VEL
LIN {X 0,Y 108.042,Z 449.732,A -85,B 0,C 180,E1 -26858.687,E2 -26858.687} C_VEL
LIN {X 0,Y 103.999,Z 451.817,A -85,B 0,C 180,E1 -26862.495,E2 -26862.495} C_VEL
LIN {X 0,Y 100.986,Z 453.046,A -85,B 0,C 180,E1 -26865.899,E2 -26865.899} C_VEL
LIN {X 0,Y 98.098,Z 453.885,A -85,B 0,C 180,E1 -26869.852,E2 -26869.852} C_VEL
LIN {X 0,Y 95.674,Z 454.155,A -85,B 0,C 180,E1 -26874.01,E2 -26874.01} C_VEL
LIN {X 0,Y 93.717,Z 453.818,A -85,B 0,C 180,E1 -26878.337,E2 -26878.337} C_VEL
LIN {X 0,Y 92.243,Z 452.96,A -85,B 0,C 180,E1 -26882.798,E2 -26882.798} C_VEL
LIN {X 0,Y 91.34,Z 451.574,A -85,B 0,C 180,E1 -26887.375,E2 -26887.375} C_VEL
LIN {X 0,Y 90.896,Z 448.427,A -85,B 0,C 180,E1 -26894.3,E2 -26894.3} C_VEL
LIN {X 0,Y 91.499,Z 443.945,A -85,B 0,C 180,E1 -26901.164,E2 -26901.164} C_VEL
LIN {X 0,Y 92.763,Z 438.929,A -85,B 0,C 180,E1 -26906.743,E2 -26906.743} C_VEL
LIN {X 0,Y 94.54,Z 432.576,A -85,B 0,C 180,E1 -26912.131,E2 -26912.131} C_VEL
LIN {X 0,Y 96.392,Z 426.375,A -85,B 0,C 180,E1 -26916.28,E2 -26916.28} C_VEL
LIN {X 0,Y 98.401,Z 419.854,A -85,B 0,C 180,E1 -26919.767,E2 -26919.767} C_VEL
LIN {X 0,Y 100.477,Z 412.764,A -85,B 0,C 180,E1 -26922.81,E2 -26922.81} C_VEL
LIN {X 0,Y 102.392,Z 405.604,A -85,B 0,C 180,E1 -26925.278,E2 -26925.278} C_VEL
LIN {X 0,Y 104.505,Z 396.821,A -85,B 0,C 180,E1 -26927.616,E2 -26927.616} C_VEL
LIN {X 0,Y 106.108,Z 388.402,A -85,B 0,C 180,E1 -26929.341,E2 -26929.341} C_VEL
LIN {X 0,Y 107.392,Z 379.201,A -85,B 0,C 180,E1 -26930.745,E2 -26930.745} C_VEL
LIN {X 0,Y 108.378,Z 369.776,A -85,B 0,C 180,E1 -26931.679,E2 -26931.679} C_VEL
LIN {X 0,Y 110.151,Z 339.881,A -85,B 0,C 180,E1 -26933.519,E2 -26933.519} C_VEL
LIN {X 0,Y 105.136,Z 328.59,A -85,B 0,C 180,E1 -26936.291,E2 -26936.291} C_VEL
LIN {X 0,Y 100.488,Z 320.326,A -85,B 0,C 180,E1 -26938.999,E2 -26938.999} C_VEL
LIN {X 0,Y 96.375,Z 313.638,A -85,B 0,C 180,E1 -26941.645,E2 -26941.645} C_VEL
LIN {X 0,Y 94.174,Z 310.624,A -85,B 0,C 180,E1 -26943.144,E2 -26943.144} C_VEL
LIN {X 0,Y 93.613,Z 308.625,A -85,B 0,C 180,E1 -26943.784,E2 -26943.784} C_VEL
LIN {X 0,Y 93.509,Z 308.645,A -85,B 0,C 180,E1 -26952.566,E2 -26952.566} C_VEL
LIN {X 0,Y 93.515,Z 308.647,A -85,B 0,C 180,E1 -26958.725,E2 -26958.725} C_VEL
LIN {X 0,Y 93.572,Z 308.638,A -85,B 0,C 180,E1 -26965.711,E2 -26965.711} C_VEL
LIN {X 0,Y 93.671,Z 308.621,A -85,B 0,C 180,E1 -26974.205,E2 -26974.205} C_VEL
LIN {X 0,Y 94.657,Z 308.499,A -85,B 0,C 180,E1 -26984.846,E2 -26984.846} C_VEL
LIN {X 0,Y 97.47,Z 308.142,A -85,B 0,C 180,E1 -26992.766,E2 -26992.766} C_VEL
LIN {X 0,Y 98.174,Z 308.075,A -85,B 0,C 180,E1 -26993.722,E2 -26993.722} C_VEL
LIN {X 0,Y 98.898,Z 313.949,A -85,B 0,C 180,E1 -26994.472,E2 -26994.472} C_VEL
LIN {X 0,Y 101.098,Z 361.098,A -85,B 0,C 180,E1 -27001.88,E2 -27001.88} C_VEL
LIN {X 0,Y 101.407,Z 373.569,A -85,B 0,C 180,E1 -27004.124,E2 -27004.124} C_VEL
LIN {X 0,Y 101.522,Z 384.727,A -85,B 0,C 180,E1 -27006.879,E2 -27006.879} C_VEL
LIN {X 0,Y 101.774,Z 394.064,A -85,B 0,C 180,E1 -27009.931,E2 -27009.931} C_VEL
LIN {X 0,Y 101.884,Z 403.796,A -85,B 0,C 180,E1 -27014.187,E2 -27014.187} C_VEL
LIN {X 0,Y 102.66,Z 412.748,A -85,B 0,C 180,E1 -27018.989,E2 -27018.989} C_VEL
LIN {X 0,Y 104.668,Z 421.825,A -85,B 0,C 180,E1 -27024.826,E2 -27024.826} C_VEL
LIN {X 0,Y 108.144,Z 429.69,A -85,B 0,C 180,E1 -27030.255,E2 -27030.255} C_VEL
LIN {X 0,Y 113.865,Z 437.456,A -85,B 0,C 180,E1 -27035.912,E2 -27035.912} C_VEL
LIN {X 0,Y 120.013,Z 443.014,A -85,B 0,C 180,E1 -27040.115,E2 -27040.115} C_VEL
LIN {X 0,Y 124.562,Z 446.256,A -85,B 0,C 180,E1 -27042.626,E2 -27042.626} C_VEL
LIN {X 0,Y 126.939,Z 447.718,A -85,B 0,C 180,E1 -27043.966,E2 -27043.966} C_VEL
LIN {X 0,Y 117.99,Z 442.924,A -85,B 0,C 180,E1 -27049.064,E2 -27049.064} C_VEL
LIN {X 0,Y 112.498,Z 438.515,A -85,B 0,C 180,E1 -27053.594,E2 -27053.594} C_VEL
LIN {X 0,Y 107.603,Z 432.098,A -85,B 0,C 180,E1 -27060.045,E2 -27060.045} C_VEL
LIN {X 0,Y 105.66,Z 427.79,A -85,B 0,C 180,E1 -27064.184,E2 -27064.184} C_VEL
LIN {X 0,Y 102.571,Z 431.786,A -85,B 0,C 180,E1 -27065.725,E2 -27065.725} C_VEL
LIN {X 0,Y 98.447,Z 438.132,A -85,B 0,C 180,E1 -27069.087,E2 -27069.087} C_VEL
LIN {X 0,Y 94.935,Z 444.688,A -85,B 0,C 180,E1 -27073.881,E2 -27073.881} C_VEL
LIN {X 0,Y 92.72,Z 450.002,A -85,B 0,C 180,E1 -27079.076,E2 -27079.076} C_VEL
LIN {X 0,Y 91.79,Z 453.476,A -85,B 0,C 180,E1 -27083.404,E2 -27083.404} C_VEL
LIN {X 0,Y 91.498,Z 455.975,A -85,B 0,C 180,E1 -27087.132,E2 -27087.132} C_VEL
LIN {X 0,Y 91.424,Z 458.328,A -85,B 0,C 180,E1 -27091.704,E2 -27091.704} C_VEL
LIN {X 0,Y 91.515,Z 460.744,A -85,B 0,C 180,E1 -27098.834,E2 -27098.834} C_VEL
LIN {X 0,Y 92.179,Z 461.614,A -85,B 0,C 180,E1 -27103.221,E2 -27103.221} C_VEL
LIN {X 0,Y 93.384,Z 461.916,A -85,B 0,C 180,E1 -27107.519,E2 -27107.519} C_VEL
LIN {X 0,Y 95.104,Z 461.777,A -85,B 0,C 180,E1 -27111.683,E2 -27111.683} C_VEL
LIN {X 0,Y 97.278,Z 461.202,A -85,B 0,C 180,E1 -27115.688,E2 -27115.688} C_VEL
LIN {X 0,Y 100.069,Z 460.161,A -85,B 0,C 180,E1 -27119.446,E2 -27119.446} C_VEL
LIN {X 0,Y 105.047,Z 457.544,A -85,B 0,C 180,E1 -27124.657,E2 -27124.657} C_VEL
LIN {X 0,Y 110.791,Z 453.691,A -85,B 0,C 180,E1 -27129.371,E2 -27129.371} C_VEL
LIN {X 0,Y 117.404,Z 448.486,A -85,B 0,C 180,E1 -27133.503,E2 -27133.503} C_VEL
LIN {X 0,Y 124.525,Z 441.683,A -85,B 0,C 180,E1 -27137.197,E2 -27137.197} C_VEL
LIN {X 0,Y 130.881,Z 434.279,A -85,B 0,C 180,E1 -27139.923,E2 -27139.923} C_VEL
LIN {X 0,Y 136.179,Z 427.005,A -85,B 0,C 180,E1 -27141.908,E2 -27141.908} C_VEL
LIN {X 0,Y 140.999,Z 419.237,A -85,B 0,C 180,E1 -27143.488,E2 -27143.488} C_VEL
LIN {X 0,Y 142.759,Z 416.132,A -85,B 0,C 180,E1 -27144.025,E2 -27144.025} C_VEL
LIN {X 0,Y 145.733,Z 409.532,A -85,B 0,C 180,E1 -27145.255,E2 -27145.255} C_VEL
LIN {X 0,Y 147.771,Z 402.775,A -85,B 0,C 180,E1 -27146.636,E2 -27146.636} C_VEL
LIN {X 0,Y 149.156,Z 395.825,A -85,B 0,C 180,E1 -27148.024,E2 -27148.024} C_VEL
LIN {X 0,Y 150.125,Z 388.641,A -85,B 0,C 180,E1 -27149.271,E2 -27149.271} C_VEL
LIN {X 0,Y 148.849,Z 382.311,A -85,B 0,C 180,E1 -27152.161,E2 -27152.161} C_VEL
LIN {X 0,Y 147.174,Z 376.731,A -85,B 0,C 180,E1 -27155.257,E2 -27155.257} C_VEL
LIN {X 0,Y 146.018,Z 373.279,A -85,B 0,C 180,E1 -27157.718,E2 -27157.718} C_VEL
LIN {X 0,Y 143.959,Z 369.265,A -85,B 0,C 180,E1 -27162.593,E2 -27162.593} C_VEL
LIN {X 0,Y 142.456,Z 365.715,A -85,B 0,C 180,E1 -27171.058,E2 -27171.058} C_VEL
LIN {X 0,Y 142.653,Z 365.608,A -85,B 0,C 180,E1 -27174.717,E2 -27174.717} C_VEL
LIN {X 0,Y 144.107,Z 369.151,A -85,B 0,C 180,E1 -27181.388,E2 -27181.388} C_VEL
LIN {X 0,Y 145.921,Z 373.261,A -85,B 0,C 180,E1 -27186.039,E2 -27186.039} C_VEL
LIN {X 0,Y 147.84,Z 377.654,A -85,B 0,C 180,E1 -27189.741,E2 -27189.741} C_VEL
LIN {X 0,Y 149.724,Z 382.849,A -85,B 0,C 180,E1 -27193.264,E2 -27193.264} C_VEL
LIN {X 0,Y 150.271,Z 384.494,A -85,B 0,C 180,E1 -27194.215,E2 -27194.215} C_VEL
LIN {X 0,Y 150.001,Z 386.39,A -85,B 0,C 180,E1 -27194.576,E2 -27194.576} C_VEL
LIN {X 0,Y 147.051,Z 395.63,A -85,B 0,C 180,E1 -27195.418,E2 -27195.418} C_VEL
LIN {X 0,Y 143.033,Z 405.285,A -85,B 0,C 180,E1 -27196.642,E2 -27196.642} C_VEL
LIN {X 0,Y 138.585,Z 413.747,A -85,B 0,C 180,E1 -27198.038,E2 -27198.038} C_VEL
LIN {X 0,Y 133.512,Z 421.733,A -85,B 0,C 180,E1 -27199.793,E2 -27199.793} C_VEL
LIN {X 0,Y 127.488,Z 429.62,A -85,B 0,C 180,E1 -27202.109,E2 -27202.109} C_VEL
LIN {X 0,Y 120.413,Z 437.058,A -85,B 0,C 180,E1 -27205.222,E2 -27205.222} C_VEL
LIN {X 0,Y 115.221,Z 441.656,A -85,B 0,C 180,E1 -27207.818,E2 -27207.818} C_VEL
LIN {X 0,Y 110.535,Z 445.301,A -85,B 0,C 180,E1 -27210.559,E2 -27210.559} C_VEL
LIN {X 0,Y 105.708,Z 448.493,A -85,B 0,C 180,E1 -27213.793,E2 -27213.793} C_VEL
LIN {X 0,Y 99.446,Z 451.736,A -85,B 0,C 180,E1 -27218.979,E2 -27218.979} C_VEL
LIN {X 0,Y 95.746,Z 453.223,A -85,B 0,C 180,E1 -27222.776,E2 -27222.776} C_VEL
LIN {X 0,Y 92.5,Z 454.148,A -85,B 0,C 180,E1 -27226.86,E2 -27226.86} C_VEL
LIN {X 0,Y 89.376,Z 454.487,A -85,B 0,C 180,E1 -27231.819,E2 -27231.819} C_VEL
LIN {X 0,Y 87.451,Z 454.216,A -85,B 0,C 180,E1 -27235.769,E2 -27235.769} C_VEL
LIN {X 0,Y 85.678,Z 453.467,A -85,B 0,C 180,E1 -27240.518,E2 -27240.518} C_VEL
LIN {X 0,Y 84.388,Z 451.884,A -85,B 0,C 180,E1 -27246.32,E2 -27246.32} C_VEL
LIN {X 0,Y 83.8,Z 449.159,A -85,B 0,C 180,E1 -27252.931,E2 -27252.931} C_VEL
LIN {X 0,Y 83.962,Z 446.4,A -85,B 0,C 180,E1 -27257.922,E2 -27257.922} C_VEL
LIN {X 0,Y 84.812,Z 442.235,A -85,B 0,C 180,E1 -27263.767,E2 -27263.767} C_VEL
LIN {X 0,Y 86.143,Z 437.631,A -85,B 0,C 180,E1 -27268.832,E2 -27268.832} C_VEL
LIN {X 0,Y 87.752,Z 432.402,A -85,B 0,C 180,E1 -27273.445,E2 -27273.445} C_VEL
LIN {X 0,Y 89.773,Z 426.103,A -85,B 0,C 180,E1 -27277.875,E2 -27277.875} C_VEL
LIN {X 0,Y 91.933,Z 419.472,A -85,B 0,C 180,E1 -27281.577,E2 -27281.577} C_VEL
LIN {X 0,Y 94.183,Z 412.358,A -85,B 0,C 180,E1 -27284.727,E2 -27284.727} C_VEL
LIN {X 0,Y 96.413,Z 404.436,A -85,B 0,C 180,E1 -27287.5,E2 -27287.5} C_VEL
LIN {X 0,Y 98.505,Z 395.863,A -85,B 0,C 180,E1 -27289.81,E2 -27289.81} C_VEL
LIN {X 0,Y 100.28,Z 386.752,A -85,B 0,C 180,E1 -27291.662,E2 -27291.662} C_VEL
LIN {X 0,Y 101.987,Z 374.679,A -85,B 0,C 180,E1 -27293.338,E2 -27293.338} C_VEL
LIN {X 0,Y 103.239,Z 357.583,A -85,B 0,C 180,E1 -27294.56,E2 -27294.56} C_VEL
LIN {X 0,Y 104.216,Z 341.798,A -85,B 0,C 180,E1 -27295.529,E2 -27295.529} C_VEL
LIN {X 0,Y 98.792,Z 329.893,A -85,B 0,C 180,E1 -27298.884,E2 -27298.884} C_VEL
LIN {X 0,Y 93.453,Z 320.943,A -85,B 0,C 180,E1 -27302.462,E2 -27302.462} C_VEL
LIN {X 0,Y 91.456,Z 317.73,A -85,B 0,C 180,E1 -27303.953,E2 -27303.953} C_VEL
LIN {X 0,Y 89.211,Z 314.298,A -85,B 0,C 180,E1 -27305.737,E2 -27305.737} C_VEL
LIN {X 0,Y 87.214,Z 312,A -85,B 0,C 180,E1 -27307.361,E2 -27307.361} C_VEL
LIN {X 0,Y 86.412,Z 309.525,A -85,B 0,C 180,E1 -27308.356,E2 -27308.356} C_VEL
LIN {X 0,Y 86.433,Z 309.524,A -85,B 0,C 180,E1 -27312.986,E2 -27312.986} C_VEL
LIN {X 0,Y 86.438,Z 309.524,A -85,B 0,C 180,E1 -27319.446,E2 -27319.446} C_VEL
LIN {X 0,Y 86.515,Z 309.519,A -85,B 0,C 180,E1 -27325.364,E2 -27325.364} C_VEL
LIN {X 0,Y 86.582,Z 309.508,A -85,B 0,C 180,E1 -27333.241,E2 -27333.241} C_VEL
LIN {X 0,Y 87.835,Z 309.355,A -85,B 0,C 180,E1 -27346.127,E2 -27346.127} C_VEL
LIN {X 0,Y 89.301,Z 309.164,A -85,B 0,C 180,E1 -27350.959,E2 -27350.959} C_VEL
LIN {X 0,Y 92.063,Z 308.806,A -85,B 0,C 180,E1 -27355.836,E2 -27355.836} C_VEL
LIN {X 0,Y 92.739,Z 314.626,A -85,B 0,C 180,E1 -27356.682,E2 -27356.682} C_VEL
LIN {X 0,Y 95.465,Z 361.516,A -85,B 0,C 180,E1 -27364.5,E2 -27364.5} C_VEL
LIN {X 0,Y 95.882,Z 373.451,A -85,B 0,C 180,E1 -27366.854,E2 -27366.854} C_VEL
LIN {X 0,Y 96.148,Z 383.323,A -85,B 0,C 180,E1 -27369.468,E2 -27369.468} C_VEL
LIN {X 0,Y 96.474,Z 392.538,A -85,B 0,C 180,E1 -27372.637,E2 -27372.637} C_VEL
LIN {X 0,Y 96.768,Z 401.87,A -85,B 0,C 180,E1 -27376.902,E2 -27376.902} C_VEL
LIN {X 0,Y 97.83,Z 411.197,A -85,B 0,C 180,E1 -27382.171,E2 -27382.171} C_VEL
LIN {X 0,Y 100.335,Z 420.436,A -85,B 0,C 180,E1 -27388.23,E2 -27388.23} C_VEL
LIN {X 0,Y 105.155,Z 429.548,A -85,B 0,C 180,E1 -27394.631,E2 -27394.631} C_VEL
LIN {X 0,Y 111.762,Z 437.339,A -85,B 0,C 180,E1 -27400.146,E2 -27400.146} C_VEL
LIN {X 0,Y 116.582,Z 441.47,A -85,B 0,C 180,E1 -27403.14,E2 -27403.14} C_VEL
LIN {X 0,Y 117.703,Z 442.459,A -85,B 0,C 180,E1 -27404.232,E2 -27404.232} C_VEL
LIN {X 0,Y 109.399,Z 436.413,A -85,B 0,C 180,E1 -27410.026,E2 -27410.026} C_VEL
LIN {X 0,Y 104.816,Z 431.394,A -85,B 0,C 180,E1 -27415.025,E2 -27415.025} C_VEL
LIN {X 0,Y 101.087,Z 424.461,A -85,B 0,C 180,E1 -27421.729,E2 -27421.729} C_VEL
LIN {X 0,Y 97.533,Z 428.656,A -85,B 0,C 180,E1 -27423.232,E2 -27423.232} C_VEL
LIN {X 0,Y 92.922,Z 435.478,A -85,B 0,C 180,E1 -27426.604,E2 -27426.604} C_VEL
LIN {X 0,Y 88.82,Z 442.591,A -85,B 0,C 180,E1 -27431.547,E2 -27431.547} C_VEL
LIN {X 0,Y 86.597,Z 447.225,A -85,B 0,C 180,E1 -27435.907,E2 -27435.907} C_VEL
LIN {X 0,Y 84.763,Z 452.76,A -85,B 0,C 180,E1 -27442.855,E2 -27442.855} C_VEL
LIN {X 0,Y 84.484,Z 456.846,A -85,B 0,C 180,E1 -27449.999,E2 -27449.999} C_VEL
LIN {X 0,Y 84.253,Z 458.815,A -85,B 0,C 180,E1 -27454.784,E2 -27454.784} C_VEL
LIN {X 0,Y 84.493,Z 460.28,A -85,B 0,C 180,E1 -27459.575,E2 -27459.575} C_VEL
LIN {X 0,Y 85.27,Z 461.161,A -85,B 0,C 180,E1 -27464.315,E2 -27464.315} C_VEL
LIN {X 0,Y 86.638,Z 461.545,A -85,B 0,C 180,E1 -27468.933,E2 -27468.933} C_VEL
LIN {X 0,Y 88.534,Z 461.492,A -85,B 0,C 180,E1 -27473.384,E2 -27473.384} C_VEL
LIN {X 0,Y 90.916,Z 461.004,A -85,B 0,C 180,E1 -27477.632,E2 -27477.632} C_VEL
LIN {X 0,Y 93.937,Z 459.987,A -85,B 0,C 180,E1 -27481.581,E2 -27481.581} C_VEL
LIN {X 0,Y 99.296,Z 457.523,A -85,B 0,C 180,E1 -27486.985,E2 -27486.985} C_VEL
LIN {X 0,Y 105.407,Z 453.775,A -85,B 0,C 180,E1 -27491.816,E2 -27491.816} C_VEL
LIN {X 0,Y 109.989,Z 450.598,A -85,B 0,C 180,E1 -27494.657,E2 -27494.657} C_VEL
LIN {X 0,Y 116.044,Z 445.592,A -85,B 0,C 180,E1 -27497.875,E2 -27497.875} C_VEL
LIN {X 0,Y 121.268,Z 440.511,A -85,B 0,C 180,E1 -27500.355,E2 -27500.355} C_VEL
LIN {X 0,Y 126.45,Z 434.87,A -85,B 0,C 180,E1 -27502.372,E2 -27502.372} C_VEL
LIN {X 0,Y 131.936,Z 427.779,A -85,B 0,C 180,E1 -27504.324,E2 -27504.324} C_VEL
LIN {X 0,Y 136.912,Z 420.236,A -85,B 0,C 180,E1 -27505.865,E2 -27505.865} C_VEL
LIN {X 0,Y 141.295,Z 412.35,A -85,B 0,C 180,E1 -27507.072,E2 -27507.072} C_VEL
LIN {X 0,Y 145.052,Z 404.233,A -85,B 0,C 180,E1 -27507.98,E2 -27507.98} C_VEL
LIN {X 0,Y 148.398,Z 394.893,A -85,B 0,C 180,E1 -27508.805,E2 -27508.805} C_VEL
LIN {X 0,Y 150.125,Z 388.641,A -85,B 0,C 180,E1 -27509.271,E2 -27509.271} C_VEL
LIN {X 0,Y 150.132,Z 385.967,A -85,B 0,C 180,E1 -27509.952,E2 -27509.952} C_VEL
LIN {X 0,Y 149.484,Z 383.485,A -85,B 0,C 180,E1 -27511.228,E2 -27511.228} C_VEL
LIN {X 0,Y 148.022,Z 381.515,A -85,B 0,C 180,E1 -27513.302,E2 -27513.302} C_VEL
LIN {X 0,Y 144.104,Z 379.4,A -85,B 0,C 180,E1 -27519.073,E2 -27519.073} C_VEL
LIN {X 0,Y 143.387,Z 378.182,A -85,B 0,C 180,E1 -27520.747,E2 -27520.747} C_VEL
LIN {X 0,Y 142.653,Z 376.125,A -85,B 0,C 180,E1 -27523.167,E2 -27523.167} C_VEL
LIN {X 0,Y 141.483,Z 372.686,A -85,B 0,C 180,E1 -27531.421,E2 -27531.421} C_VEL
LIN {X 0,Y 141.633,Z 372.672,A -85,B 0,C 180,E1 -27534.487,E2 -27534.487} C_VEL
LIN {X 0,Y 142.873,Z 376.398,A -85,B 0,C 180,E1 -27541.4,E2 -27541.4} C_VEL
LIN {X 0,Y 144.15,Z 380.195,A -85,B 0,C 180,E1 -27545.587,E2 -27545.587} C_VEL
LIN {X 0,Y 145.412,Z 384.045,A -85,B 0,C 180,E1 -27548.94,E2 -27548.94} C_VEL
LIN {X 0,Y 146.631,Z 388.515,A -85,B 0,C 180,E1 -27552.112,E2 -27552.112} C_VEL
LIN {X 0,Y 143.681,Z 397.373,A -85,B 0,C 180,E1 -27553.025,E2 -27553.025} C_VEL
LIN {X 0,Y 140.27,Z 405.23,A -85,B 0,C 180,E1 -27553.985,E2 -27553.985} C_VEL
LIN {X 0,Y 136.491,Z 412.378,A -85,B 0,C 180,E1 -27555.075,E2 -27555.075} C_VEL
LIN {X 0,Y 131.918,Z 419.603,A -85,B 0,C 180,E1 -27556.474,E2 -27556.474} C_VEL
LIN {X 0,Y 127.476,Z 425.664,A -85,B 0,C 180,E1 -27558.007,E2 -27558.007} C_VEL
LIN {X 0,Y 121.282,Z 432.73,A -85,B 0,C 180,E1 -27560.334,E2 -27560.334} C_VEL
LIN {X 0,Y 114.641,Z 439.022,A -85,B 0,C 180,E1 -27563.139,E2 -27563.139} C_VEL
LIN {X 0,Y 107.34,Z 444.809,A -85,B 0,C 180,E1 -27566.89,E2 -27566.89} C_VEL
LIN {X 0,Y 101.739,Z 448.377,A -85,B 0,C 180,E1 -27570.291,E2 -27570.291} C_VEL
LIN {X 0,Y 94.909,Z 451.8,A -85,B 0,C 180,E1 -27575.459,E2 -27575.459} C_VEL
LIN {X 0,Y 90.841,Z 453.39,A -85,B 0,C 180,E1 -27579.317,E2 -27579.317} C_VEL
LIN {X 0,Y 87.192,Z 454.353,A -85,B 0,C 180,E1 -27583.496,E2 -27583.496} C_VEL
LIN {X 0,Y 83.076,Z 454.824,A -85,B 0,C 180,E1 -27589.559,E2 -27589.559} C_VEL
LIN {X 0,Y 79.279,Z 453.975,A -85,B 0,C 180,E1 -27597.868,E2 -27597.868} C_VEL
LIN {X 0,Y 77.432,Z 452.174,A -85,B 0,C 180,E1 -27605.136,E2 -27605.136} C_VEL
LIN {X 0,Y 76.765,Z 449.891,A -85,B 0,C 180,E1 -27611.312,E2 -27611.312} C_VEL
LIN {X 0,Y 77.013,Z 445.661,A -85,B 0,C 180,E1 -27619.485,E2 -27619.485} C_VEL
LIN {X 0,Y 78.557,Z 439.941,A -85,B 0,C 180,E1 -27627.437,E2 -27627.437} C_VEL
LIN {X 0,Y 80.51,Z 433.684,A -85,B 0,C 180,E1 -27633.755,E2 -27633.755} C_VEL
LIN {X 0,Y 82.642,Z 427.565,A -85,B 0,C 180,E1 -27638.56,E2 -27638.56} C_VEL
LIN {X 0,Y 85.246,Z 420.114,A -85,B 0,C 180,E1 -27643.105,E2 -27643.105} C_VEL
LIN {X 0,Y 87.888,Z 412.32,A -85,B 0,C 180,E1 -27646.758,E2 -27646.758} C_VEL
LIN {X 0,Y 90.451,Z 403.702,A -85,B 0,C 180,E1 -27649.874,E2 -27649.874} C_VEL
LIN {X 0,Y 92.96,Z 393.622,A -85,B 0,C 180,E1 -27652.603,E2 -27652.603} C_VEL
LIN {X 0,Y 95.13,Z 381.773,A -85,B 0,C 180,E1 -27654.753,E2 -27654.753} C_VEL
LIN {X 0,Y 96.36,Z 372.441,A -85,B 0,C 180,E1 -27655.832,E2 -27655.832} C_VEL
LIN {X 0,Y 98.352,Z 343.798,A -85,B 0,C 180,E1 -27657.784,E2 -27657.784} C_VEL
LIN {X 0,Y 93.599,Z 333.185,A -85,B 0,C 180,E1 -27661.12,E2 -27661.12} C_VEL
LIN {X 0,Y 88.817,Z 325.03,A -85,B 0,C 180,E1 -27664.759,E2 -27664.759} C_VEL
LIN {X 0,Y 85.439,Z 319.732,A -85,B 0,C 180,E1 -27667.68,E2 -27667.68} C_VEL
LIN {X 0,Y 83.181,Z 316.518,A -85,B 0,C 180,E1 -27669.823,E2 -27669.823} C_VEL
LIN {X 0,Y 82.417,Z 315.383,A -85,B 0,C 180,E1 -27670.604,E2 -27670.604} C_VEL
LIN {X 0,Y 80.364,Z 313.168,A -85,B 0,C 180,E1 -27672.707,E2 -27672.707} C_VEL
LIN {X 0,Y 79.477,Z 310.97,A -85,B 0,C 180,E1 -27673.868,E2 -27673.868} C_VEL
LIN {X 0,Y 79.35,Z 310.404,A -85,B 0,C 180,E1 -27674.23,E2 -27674.23} C_VEL
LIN {X 0,Y 79.369,Z 310.409,A -85,B 0,C 180,E1 -27682.84,E2 -27682.84} C_VEL
LIN {X 0,Y 79.476,Z 310.396,A -85,B 0,C 180,E1 -27692.166,E2 -27692.166} C_VEL
LIN {X 0,Y 80.356,Z 310.274,A -85,B 0,C 180,E1 -27704.172,E2 -27704.172} C_VEL
LIN {X 0,Y 84.532,Z 309.741,A -85,B 0,C 180,E1 -27716.112,E2 -27716.112} C_VEL
LIN {X 0,Y 86.108,Z 309.558,A -85,B 0,C 180,E1 -27718.296,E2 -27718.296} C_VEL
LIN {X 0,Y 86.752,Z 315.711,A -85,B 0,C 180,E1 -27719.304,E2 -27719.304} C_VEL
LIN {X 0,Y 90.101,Z 360.525,A -85,B 0,C 180,E1 -27727.296,E2 -27727.296} C_VEL
LIN {X 0,Y 90.685,Z 372.493,A -85,B 0,C 180,E1 -27729.775,E2 -27729.775} C_VEL
LIN {X 0,Y 90.991,Z 381.661,A -85,B 0,C 180,E1 -27732.278,E2 -27732.278} C_VEL
LIN {X 0,Y 91.391,Z 389.703,A -85,B 0,C 180,E1 -27735.111,E2 -27735.111} C_VEL
LIN {X 0,Y 91.966,Z 399.317,A -85,B 0,C 180,E1 -27739.721,E2 -27739.721} C_VEL
LIN {X 0,Y 92.8,Z 406.148,A -85,B 0,C 180,E1 -27743.56,E2 -27743.56} C_VEL
LIN {X 0,Y 94.764,Z 414.287,A -85,B 0,C 180,E1 -27748.834,E2 -27748.834} C_VEL
LIN {X 0,Y 99.399,Z 424.372,A -85,B 0,C 180,E1 -27755.698,E2 -27755.698} C_VEL
LIN {X 0,Y 105.907,Z 432.81,A -85,B 0,C 180,E1 -27761.59,E2 -27761.59} C_VEL
LIN {X 0,Y 107.886,Z 434.772,A -85,B 0,C 180,E1 -27762.948,E2 -27762.948} C_VEL
LIN {X 0,Y 108.911,Z 435.934,A -85,B 0,C 180,E1 -27764.778,E2 -27764.778} C_VEL
LIN {X 0,Y 102.32,Z 429.886,A -85,B 0,C 180,E1 -27770.484,E2 -27770.484} C_VEL
LIN {X 0,Y 98.738,Z 424.975,A -85,B 0,C 180,E1 -27775.289,E2 -27775.289} C_VEL
LIN {X 0,Y 96.732,Z 420.954,A -85,B 0,C 180,E1 -27779.127,E2 -27779.127} C_VEL
LIN {X 0,Y 92.821,Z 425.421,A -85,B 0,C 180,E1 -27780.517,E2 -27780.517} C_VEL
LIN {X 0,Y 88.749,Z 431.018,A -85,B 0,C 180,E1 -27782.912,E2 -27782.912} C_VEL
LIN {X 0,Y 84.564,Z 437.43,A -85,B 0,C 180,E1 -27786.775,E2 -27786.775} C_VEL
LIN {X 0,Y 80.923,Z 443.976,A -85,B 0,C 180,E1 -27792.303,E2 -27792.303} C_VEL
LIN {X 0,Y 78.938,Z 448.354,A -85,B 0,C 180,E1 -27797.138,E2 -27797.138} C_VEL
LIN {X 0,Y 77.77,Z 452.026,A -85,B 0,C 180,E1 -27802.208,E2 -27802.208} C_VEL
LIN {X 0,Y 77.416,Z 456.209,A -85,B 0,C 180,E1 -27809.999,E2 -27809.999} C_VEL
LIN {X 0,Y 77.195,Z 458.269,A -85,B 0,C 180,E1 -27815.223,E2 -27815.223} C_VEL
LIN {X 0,Y 77.492,Z 459.779,A -85,B 0,C 180,E1 -27820.45,E2 -27820.45} C_VEL
LIN {X 0,Y 78.409,Z 460.703,A -85,B 0,C 180,E1 -27825.598,E2 -27825.598} C_VEL
LIN {X 0,Y 79.959,Z 461.174,A -85,B 0,C 180,E1 -27830.583,E2 -27830.583} C_VEL
LIN {X 0,Y 82.037,Z 461.207,A -85,B 0,C 180,E1 -27835.361,E2 -27835.361} C_VEL
LIN {X 0,Y 84.678,Z 460.786,A -85,B 0,C 180,E1 -27839.865,E2 -27839.865} C_VEL
LIN {X 0,Y 87.958,Z 459.79,A -85,B 0,C 180,E1 -27844.007,E2 -27844.007} C_VEL
LIN {X 0,Y 91.7,Z 458.31,A -85,B 0,C 180,E1 -27847.815,E2 -27847.815} C_VEL
LIN {X 0,Y 97.959,Z 455.175,A -85,B 0,C 180,E1 -27852.965,E2 -27852.965} C_VEL
LIN {X 0,Y 105.061,Z 450.762,A -85,B 0,C 180,E1 -27857.377,E2 -27857.377} C_VEL
LIN {X 0,Y 111.58,Z 445.75,A -85,B 0,C 180,E1 -27860.657,E2 -27860.657} C_VEL
LIN {X 0,Y 118.971,Z 438.813,A -85,B 0,C 180,E1 -27863.815,E2 -27863.815} C_VEL
LIN {X 0,Y 123.653,Z 433.766,A -85,B 0,C 180,E1 -27865.5,E2 -27865.5} C_VEL
LIN {X 0,Y 129.402,Z 426.515,A -85,B 0,C 180,E1 -27867.332,E2 -27867.332} C_VEL
LIN {X 0,Y 134.577,Z 418.779,A -85,B 0,C 180,E1 -27868.776,E2 -27868.776} C_VEL
LIN {X 0,Y 138.996,Z 410.866,A -85,B 0,C 180,E1 -27869.877,E2 -27869.877} C_VEL
LIN {X 0,Y 142.969,Z 402.232,A -85,B 0,C 180,E1 -27870.734,E2 -27870.734} C_VEL
LIN {X 0,Y 146.512,Z 391.929,A -85,B 0,C 180,E1 -27871.594,E2 -27871.594} C_VEL
LIN {X 0,Y 146.5,Z 390.62,A -85,B 0,C 180,E1 -27872.102,E2 -27872.102} C_VEL
LIN {X 0,Y 145.254,Z 383.747,A -85,B 0,C 180,E1 -27875.785,E2 -27875.785} C_VEL
LIN {X 0,Y 144.288,Z 379.801,A -85,B 0,C 180,E1 -27878.621,E2 -27878.621} C_VEL
LIN {X 0,Y 143.387,Z 378.182,A -85,B 0,C 180,E1 -27880.747,E2 -27880.747} C_VEL
LIN {X 0,Y 142.852,Z 377.201,A -85,B 0,C 180,E1 -27882.246,E2 -27882.246} C_VEL
LIN {X 0,Y 141.997,Z 376.949,A -85,B 0,C 180,E1 -27884.591,E2 -27884.591} C_VEL
LIN {X 0,Y 140.777,Z 378.347,A -85,B 0,C 180,E1 -27888.583,E2 -27888.583} C_VEL
LIN {X 0,Y 140.223,Z 379.723,A -85,B 0,C 180,E1 -27892.684,E2 -27892.684} C_VEL
LIN {X 0,Y 140.251,Z 379.752,A -85,B 0,C 180,E1 -27893.513,E2 -27893.513} C_VEL
LIN {X 0,Y 140.296,Z 380.044,A -85,B 0,C 180,E1 -27894.821,E2 -27894.821} C_VEL
LIN {X 0,Y 140.994,Z 383.202,A -85,B 0,C 180,E1 -27900.883,E2 -27900.883} C_VEL
LIN {X 0,Y 141.771,Z 386.069,A -85,B 0,C 180,E1 -27904.255,E2 -27904.255} C_VEL
LIN {X 0,Y 142.741,Z 390.691,A -85,B 0,C 180,E1 -27908.485,E2 -27908.485} C_VEL
LIN {X 0,Y 143.029,Z 392.071,A -85,B 0,C 180,E1 -27909.562,E2 -27909.562} C_VEL
LIN {X 0,Y 142.705,Z 393.708,A -85,B 0,C 180,E1 -27909.95,E2 -27909.95} C_VEL
LIN {X 0,Y 137.991,Z 404.832,A -85,B 0,C 180,E1 -27911.175,E2 -27911.175} C_VEL
LIN {X 0,Y 133.805,Z 412.573,A -85,B 0,C 180,E1 -27912.286,E2 -27912.286} C_VEL
LIN {X 0,Y 128.452,Z 420.674,A -85,B 0,C 180,E1 -27913.796,E2 -27913.796} C_VEL
LIN {X 0,Y 123.842,Z 426.607,A -85,B 0,C 180,E1 -27915.261,E2 -27915.261} C_VEL
LIN {X 0,Y 117.814,Z 433.168,A -85,B 0,C 180,E1 -27917.362,E2 -27917.362} C_VEL
LIN {X 0,Y 111.937,Z 438.56,A -85,B 0,C 180,E1 -27919.65,E2 -27919.65} C_VEL
LIN {X 0,Y 106.259,Z 443.003,A -85,B 0,C 180,E1 -27922.188,E2 -27922.188} C_VEL
LIN {X 0,Y 100.807,Z 446.64,A -85,B 0,C 180,E1 -27924.999,E2 -27924.999} C_VEL
LIN {X 0,Y 93.153,Z 450.748,A -85,B 0,C 180,E1 -27929.818,E2 -27929.818} C_VEL
LIN {X 0,Y 86.281,Z 453.501,A -85,B 0,C 180,E1 -27935.459,E2 -27935.459} C_VEL
LIN {X 0,Y 82.208,Z 454.53,A -85,B 0,C 180,E1 -27939.7,E2 -27939.7} C_VEL
LIN {X 0,Y 76.932,Z 455.16,A -85,B 0,C 180,E1 -27946.929,E2 -27946.929} C_VEL
LIN {X 0,Y 73.062,Z 454.483,A -85,B 0,C 180,E1 -27954.751,E2 -27954.751} C_VEL
LIN {X 0,Y 71.229,Z 453.403,A -85,B 0,C 180,E1 -27960.441,E2 -27960.441} C_VEL
LIN {X 0,Y 69.777,Z 450.625,A -85,B 0,C 180,E1 -27969.359,E2 -27969.359} C_VEL
LIN {X 0,Y 69.628,Z 448.105,A -85,B 0,C 180,E1 -27975.385,E2 -27975.385} C_VEL
LIN {X 0,Y 70.129,Z 444.906,A -85,B 0,C 180,E1 -27981.355,E2 -27981.355} C_VEL
LIN {X 0,Y 71.625,Z 439.867,A -85,B 0,C 180,E1 -27988.595,E2 -27988.595} C_VEL
LIN {X 0,Y 73.786,Z 433.508,A -85,B 0,C 180,E1 -27995.467,E2 -27995.467} C_VEL
LIN {X 0,Y 76.165,Z 427.283,A -85,B 0,C 180,E1 -28000.636,E2 -28000.636} C_VEL
LIN {X 0,Y 78.631,Z 420.756,A -85,B 0,C 180,E1 -28004.891,E2 -28004.891} C_VEL
LIN {X 0,Y 81.171,Z 413.722,A -85,B 0,C 180,E1 -28008.49,E2 -28008.49} C_VEL
LIN {X 0,Y 83.711,Z 406.022,A -85,B 0,C 180,E1 -28011.551,E2 -28011.551} C_VEL
LIN {X 0,Y 86.111,Z 397.666,A -85,B 0,C 180,E1 -28014.085,E2 -28014.085} C_VEL
LIN {X 0,Y 88.046,Z 389.278,A -85,B 0,C 180,E1 -28016.026,E2 -28016.026} C_VEL
LIN {X 0,Y 89.701,Z 379.786,A -85,B 0,C 180,E1 -28017.623,E2 -28017.623} C_VEL
LIN {X 0,Y 90.921,Z 369.846,A -85,B 0,C 180,E1 -28018.684,E2 -28018.684} C_VEL
LIN {X 0,Y 92.705,Z 345.855,A -85,B 0,C 180,E1 -28020.297,E2 -28020.297} C_VEL
LIN {X 0,Y 88.889,Z 337.226,A -85,B 0,C 180,E1 -28023.341,E2 -28023.341} C_VEL
LIN {X 0,Y 83.421,Z 327.581,A -85,B 0,C 180,E1 -28028.181,E2 -28028.181} C_VEL
LIN {X 0,Y 81.533,Z 324.765,A -85,B 0,C 180,E1 -28030.052,E2 -28030.052} C_VEL
LIN {X 0,Y 79.018,Z 321.049,A -85,B 0,C 180,E1 -28032.791,E2 -28032.791} C_VEL
LIN {X 0,Y 76.816,Z 318.072,A -85,B 0,C 180,E1 -28035.445,E2 -28035.445} C_VEL
LIN {X 0,Y 76.067,Z 316.739,A -85,B 0,C 180,E1 -28036.478,E2 -28036.478} C_VEL
LIN {X 0,Y 73.652,Z 314.745,A -85,B 0,C 180,E1 -28039.724,E2 -28039.724} C_VEL
LIN {X 0,Y 72.594,Z 312.586,A -85,B 0,C 180,E1 -28041.578,E2 -28041.578} C_VEL
LIN {X 0,Y 72.311,Z 311.285,A -85,B 0,C 180,E1 -28042.267,E2 -28042.267} C_VEL
LIN {X 0,Y 72.365,Z 311.283,A -85,B 0,C 180,E1 -28050.97,E2 -28050.97} C_VEL
LIN {X 0,Y 72.542,Z 311.221,A -85,B 0,C 180,E1 -28057.219,E2 -28057.219} C_VEL
LIN {X 0,Y 77.423,Z 310.625,A -85,B 0,C 180,E1 -28076.897,E2 -28076.897} C_VEL
LIN {X 0,Y 80.486,Z 310.269,A -85,B 0,C 180,E1 -28081.267,E2 -28081.267} C_VEL
LIN {X 0,Y 81.977,Z 327.514,A -85,B 0,C 180,E1 -28084.472,E2 -28084.472} C_VEL
LIN {X 0,Y 84.985,Z 359.506,A -85,B 0,C 180,E1 -28090.437,E2 -28090.437} C_VEL
LIN {X 0,Y 85.801,Z 371.32,A -85,B 0,C 180,E1 -28093.033,E2 -28093.033} C_VEL
LIN {X 0,Y 86.306,Z 381.219,A -85,B 0,C 180,E1 -28095.967,E2 -28095.967} C_VEL
LIN {X 0,Y 86.84,Z 388.838,A -85,B 0,C 180,E1 -28098.903,E2 -28098.903} C_VEL
LIN {X 0,Y 87.802,Z 399.317,A -85,B 0,C 180,E1 -28104.297,E2 -28104.297} C_VEL
LIN {X 0,Y 89.909,Z 408.842,A -85,B 0,C 180,E1 -28110.301,E2 -28110.301} C_VEL
LIN {X 0,Y 93.908,Z 418.485,A -85,B 0,C 180,E1 -28116.794,E2 -28116.794} C_VEL
LIN {X 0,Y 101.396,Z 428.927,A -85,B 0,C 180,E1 -28123.894,E2 -28123.894} C_VEL
LIN {X 0,Y 100.674,Z 428.373,A -85,B 0,C 180,E1 -28125.724,E2 -28125.724} C_VEL
LIN {X 0,Y 94.261,Z 420.397,A -85,B 0,C 180,E1 -28133.381,E2 -28133.381} C_VEL
LIN {X 0,Y 92.754,Z 417.194,A -85,B 0,C 180,E1 -28136.352,E2 -28136.352} C_VEL
LIN {X 0,Y 88.45,Z 421.882,A -85,B 0,C 180,E1 -28137.564,E2 -28137.564} C_VEL
LIN {X 0,Y 82.621,Z 429.709,A -85,B 0,C 180,E1 -28140.717,E2 -28140.717} C_VEL
LIN {X 0,Y 77.169,Z 437.774,A -85,B 0,C 180,E1 -28145.901,E2 -28145.901} C_VEL
LIN {X 0,Y 74.258,Z 443.022,A -85,B 0,C 180,E1 -28150.654,E2 -28150.654} C_VEL
LIN {X 0,Y 72.098,Z 447.516,A -85,B 0,C 180,E1 -28155.894,E2 -28155.894} C_VEL
LIN {X 0,Y 70.766,Z 451.261,A -85,B 0,C 180,E1 -28161.432,E2 -28161.432} C_VEL
LIN {X 0,Y 70.34,Z 455.571,A -85,B 0,C 180,E1 -28169.999,E2 -28169.999} C_VEL
LIN {X 0,Y 70.141,Z 457.716,A -85,B 0,C 180,E1 -28175.749,E2 -28175.749} C_VEL
LIN {X 0,Y 70.525,Z 459.242,A -85,B 0,C 180,E1 -28181.495,E2 -28181.495} C_VEL
LIN {X 0,Y 71.604,Z 460.245,A -85,B 0,C 180,E1 -28187.124,E2 -28187.124} C_VEL
LIN {X 0,Y 73.345,Z 460.802,A -85,B 0,C 180,E1 -28192.536,E2 -28192.536} C_VEL
LIN {X 0,Y 75.656,Z 460.922,A -85,B 0,C 180,E1 -28197.675,E2 -28197.675} C_VEL
LIN {X 0,Y 78.593,Z 460.53,A -85,B 0,C 180,E1 -28202.447,E2 -28202.447} C_VEL
LIN {X 0,Y 82.163,Z 459.593,A -85,B 0,C 180,E1 -28206.78,E2 -28206.78} C_VEL
LIN {X 0,Y 86.186,Z 458.201,A -85,B 0,C 180,E1 -28210.718,E2 -28210.718} C_VEL
LIN {X 0,Y 92.892,Z 455.159,A -85,B 0,C 180,E1 -28215.95,E2 -28215.95} C_VEL
LIN {X 0,Y 100.395,Z 450.876,A -85,B 0,C 180,E1 -28220.356,E2 -28220.356} C_VEL
LIN {X 0,Y 108.162,Z 445.229,A -85,B 0,C 180,E1 -28224.027,E2 -28224.027} C_VEL
LIN {X 0,Y 115.294,Z 438.901,A -85,B 0,C 180,E1 -28226.786,E2 -28226.786} C_VEL
LIN {X 0,Y 121.261,Z 432.657,A -85,B 0,C 180,E1 -28228.745,E2 -28228.745} C_VEL
LIN {X 0,Y 126.487,Z 426.27,A -85,B 0,C 180,E1 -28230.246,E2 -28230.246} C_VEL
LIN {X 0,Y 131.815,Z 418.553,A -85,B 0,C 180,E1 -28231.609,E2 -28231.609} C_VEL
LIN {X 0,Y 136.323,Z 410.765,A -85,B 0,C 180,E1 -28232.609,E2 -28232.609} C_VEL
LIN {X 0,Y 139.857,Z 403.435,A -85,B 0,C 180,E1 -28233.304,E2 -28233.304} C_VEL
LIN {X 0,Y 142.673,Z 396.213,A -85,B 0,C 180,E1 -28233.892,E2 -28233.892} C_VEL
LIN {X 0,Y 143.095,Z 394.543,A -85,B 0,C 180,E1 -28234.148,E2 -28234.148} C_VEL
LIN {X 0,Y 142.528,Z 388.557,A -85,B 0,C 180,E1 -28237.763,E2 -28237.763} C_VEL
LIN {X 0,Y 142.109,Z 386.244,A -85,B 0,C 180,E1 -28239.483,E2 -28239.483} C_VEL
LIN {X 0,Y 141.001,Z 382.927,A -85,B 0,C 180,E1 -28243.709,E2 -28243.709} C_VEL
LIN {X 0,Y 140.196,Z 379.843,A -85,B 0,C 180,E1 -28251.341,E2 -28251.341} C_VEL
LIN {X 0,Y 140.251,Z 379.752,A -85,B 0,C 180,E1 -28253.513,E2 -28253.513} C_VEL
LIN {X 0,Y 140.306,Z 380.187,A -85,B 0,C 180,E1 -28255.094,E2 -28255.094} C_VEL
LIN {X 0,Y 140.261,Z 381.412,A -85,B 0,C 180,E1 -28256.611,E2 -28256.611} C_VEL
LIN {X 0,Y 140.033,Z 384.22,A -85,B 0,C 180,E1 -28258.76,E2 -28258.76} C_VEL
LIN {X 0,Y 139.236,Z 392.232,A -85,B 0,C 180,E1 -28263.66,E2 -28263.66} C_VEL
LIN {X 0,Y 139.334,Z 394.063,A -85,B 0,C 180,E1 -28265.176,E2 -28265.176} C_VEL
LIN {X 0,Y 139.607,Z 396.493,A -85,B 0,C 180,E1 -28267.42,E2 -28267.42} C_VEL
LIN {X 0,Y 135.46,Z 405.679,A -85,B 0,C 180,E1 -28268.429,E2 -28268.429} C_VEL
